# B&R Automation Studio project AriesV2 (part 3)

#### wbrPingSvc.c
```c
/********************************************************************
 * \copyright -- Piedmont Automation
 ********************************************************************
 * Program : wbrPingSvc
 * \file :   wbrPingSvc.c
 * \author : Blanton Radford
 * \date Created: June 22, 2015
 *******************************************************************/

#include <string.h>
// #include <bur/plctypes.h>

// #include  "wbrsprintf.h"
#include  "wbrPingSvc.h"

DINT  wbrPingSvcInit(struct wbrPingService_typ* p)
{
  p->fb.enable=  1;
  // p->fb.pHost=   (UDINT)"192.168.44.220";
  p->fb.pHost=   (UDINT)p->destIPAddr;
  p->fb.timeout= p->timeout;                                                    // If ping not successful within (timeout x 10)ms, error occurs

  p->logbookID= arlogBASE_USER_LOG_IDENT;         /// \todo   change to user net log from wbrNetSvc

  return  0;
}

static  char* errorTextLookup(UINT erNum, char* erText, UDINT erTextLen)
{
  // TODO: use table(s) in file(s) for holding error text instead of the code below

  switch(erNum)
  {
   case 32750:  wbrsnprintf(erText, erTextLen, "No response from station %%s within the specified time");
    break;
   case 32751:  wbrsnprintf(erText, erTextLen, "IP address %%s not resolvable");
    break;
   case 32752:  wbrsnprintf(erText, erTextLen, "Resource problem in system.  Could not create socket for pinging %%s");
    break;
   case 32799:  wbrsnprintf(erText, erTextLen, "System level error when pinging %%s");
    break;
   case 0xFFFE: wbrsnprintf(erText, erTextLen, "System ping function not enabled when pinging %%s");
    break;

   default:     wbrsnprintf(erText, erTextLen, "Something went wrong with error text lookup - erNum in table?");
    break;
  }

  return erText;
}

// void printErrorText(UINT erNum, char* errorText, args)  //  TODO: with variable args
// {
// }

static  void printErrorText(BOOL prependErNum, UINT erNum, char* message, UDINT msgLen, char* ipAddr)
{
  // char  erText[100]= "",      // Will contain error text with inserted format specifiers for custom arguments
        // erFmtd[100]= "";      // Will contain above text with error number prepended
  char  erText[msgLen],      // Will contain error text with inserted format specifiers for custom arguments - v0.11.0
        erFmtd[msgLen];      // Will contain above text with error number prepended

  if(prependErNum)
  {
    wbrsnprintf(erFmtd,                                                           // Used in next wbrsnprintf
              sizeof(erFmtd),
              "%d: %s",
              erNum,
              errorTextLookup(erNum, erText, sizeof(erText)));                  // Finds custom error text for error erNum

    wbrsnprintf(message,
              msgLen,
              erFmtd,                                                           // From wbrsnprintf above
              ipAddr);
    return;
  }

  // Else do not prepend error number
  wbrsnprintf(message,
            msgLen,
            errorTextLookup(erNum, erText, sizeof(erText)),                     // Finds custom error text for error erNum
            ipAddr);
  return;
}

/*! \brief Print the number of successes for debugging
    \pre   None
*/
static  char * printMsgSuccess(struct wbrPingService_typ* p)
{
  wbrsnprintf(  p->message                                                    // Print the number of successes for debugging
              , sizeof(p->message)
              , "Station %s pinged successfully %d times"
              , p->destIPPrev
              , p->count
              );
  return  p->message;
}

/*! \brief Print the number of failures for debugging
    \pre   None
*/
static  char * printMsgFailure(struct wbrPingService_typ* p)
{
  wbrsnprintf(  p->message1                                                    // Print the number of failures for debugging
              , sizeof(p->message1)
              , "Station %s ping failed %d times"
              , p->destIPPrev
              , p->count
              );
  return  p->message1;
}

DINT  wbrPingStation(struct wbrPingService_typ* p)
{
  if(!p->enable && !p->count)  return  0xFFFE;

  if(!p->enable){

    if(p->failed) requestMessageToLogDefault( (UDINT)printMsgFailure(p));
    else          requestMessageToLogDefault( (UDINT)printMsgSuccess(p));

    p->count=
        p->failed=
        p->errorStatus= 0;

    return  0xFFFE;
  }

  bgTimerCyclic(&p->retryTimer);

  if(!p->failed && p->retryTimer.IN && !p->retryTimer.Q)  return  0xFFFF;       // Return if success and the timer is running for the next attempt

  if(strcmp(p->destIPPrev, p->destIPAddr) )                                                               // new station
  {
    wbrsnprintf(p->message,                                                     // Print the number of failures for debugging
              sizeof(p->message),
              "Station %s is a new station",
              p->destIPAddr
              );
    requestMessageToLogDefault( (UDINT)p->message);

    if(p->failed) requestMessageToLogDefault( (UDINT)printMsgFailure(p));
    else          requestMessageToLogDefault( (UDINT)printMsgSuccess(p));

    p->count=
        p->failed=
        p->errorStatus= 0;
    wbrsnprintf(p->destIPPrev, sizeof(p->destIPPrev), p->destIPAddr);
  }

  p->fb.pHost=   (UDINT)p->destIPAddr;
  p->fb.timeout= p->timeout;

  IcmpPing(&p->fb);

  switch(p->fb.status)
  {
   case 0xFFFF:       //  busy
    // p->errorStatus= 0;
    return  0xFFFF;

   case 0:            //  success
    if(p->failed)                                                               // fail state changed from fail to success
    {
      requestMessageToLogDefault( (UDINT)printMsgFailure(p));
      p->count=
          p->failed=
          p->errorStatus= 0;
    }

    p->failed=  0;
    p->count++;
    bgTimerStart(&p->retryTimer, p->repeatTime);

    printMsgSuccess(p);

    if(!((p->count - 1) % p->successesToCount))
    {
      requestMessageToLogDefault( (UDINT)p->message);
    }
    return  0;

   case 32750:        // Defined error statuses
   case 32751:
   case 32752:
   case 32799:
   case 0xFFFE:
    printErrorText(1, p->fb.status, p->message, sizeof(p->message), p->destIPAddr);
    break;

   default:
    wbrsnprintf(p->message,
              sizeof(p->message),
              "%d: Should not get here when pinging IP address %s",
              p->fb.status,
              p->destIPAddr);
    break;
  }

  if(!p->failed || (p->fb.status != p->errorStatus)) //
  {
    p->errorStatus= p->fb.status;
    requestMessageToLog( (UDINT)p->message
                       , p->logbookID
                       , arlogLEVEL_INFO
                       , 55550
                       , (UDINT)&p->fb.status
                       , (UDINT)sizeof(p->fb.status)
                       );
    p->count= 0;
  }

  if(p->count == 1)
  {
    requestMessageToLog( (UDINT)"Current ping error is repeating"
                       , p->logbookID
                       , arlogLEVEL_INFO
                       , 55550
                       , (UDINT)&p->fb.status
                       , (UDINT)sizeof(p->fb.status)
                       );
  }

  p->failed=  1;
  p->count++;
  return  p->count;
}

// void  mbTCPdiag()
// {
  // slave.diag.ping.fb.pHost=   (UDINT)slave.diag.ping.destIPAddr;
  // if(slave.diag.ping.enable)   pingPeer(&slave.diag.ping, 512);
// }

DINT  wbrSQL_DT2_ISOFmtdStringFromDT(struct DTStructure * pDT, char * pDst, UDINT dstSize)
{
  return  wbrsnprintf(pDst, dstSize, "%04d-%02d-%02dT%02d:%02d:%02d",
                      pDT->year, pDT->month, pDT->day,
                      pDT->hour, pDT->minute, pDT->second);
}
```

### Library Logical/UserLibraries/wbrServices/wbrsprintf (ANSIC) - Writes user-formatted output to a string

#### wbrsprintf.h
```c
/*!
 ********************************************************************
### Library : wbrsprintf
 *  Package : WBRServices
 * \file :   wbrsprintf.h
 * \author : Blanton Radford
 * \date Created: May 3, 2016
 * \copyright -- Piedmont Automation
 *******************************************************************
 * \brief Header file for snprintf functions.
          Use of sprintf functions discouraged as snprintf is guaranteed to
          stop writing once buf_size is filled.
 ********************************************************************/

#include <stdarg.h>

/*! These are not included by default to strongly discourage the use of sprintf
    If they are uncommented, please uncomment the warning as well
*/
// #warning  "Consider using snprintf function for safety"
// int wbrvsprintf(char *s, const char *fmt, va_list ap);
// int  wbrsprintf(char *s, const char *fmt, ...);

int wbrvsnprintf(char *s, int buf_size, const char *fmt, va_list ap);
int  wbrsnprintf(char *s, int buf_size, const char *fmt, ...);
```

### Library Logical/UserLibraries/wbrServices/wbrSvcUtilities/wbrBytUtil (ANSIC)

#### wbrBytUtilities.c
```c
/*!
 ********************************************************************
### Library : wbrBytUtil
 * \file :   wbrBytUtilities.c
 * \author : Blanton Radford
 * \date Created: Friday, October 14, 2016
 * \copyright  Piedmont Automation
 ********************************************************************
 * \brief Utilities for extracting bytes from or packing bytes into words,
          ints, etc.
 ********************************************************************/

/*! \mainpage Example logbook manager to create, get info from, and write to user created logbooks using \e wbrLogSvc functions

#   A main heading

    Some text

##  A subheading

    More text

    A separator
    -----------

    Even more txt

##  See \e Files selection above for more info on the functions and how to
##  use them.
*/

#include "wbrBytUtil.h"

/*————————————————————————————————————————————————————————————————————————————*/
/*! \brief Get the high 16-bit word from a 32-bit double word
    \pre

rtyp  �(x)뿓뿓뿬  뿓뿓뿓뿓뿓뿓뾞rgument comments뿓뿓뿓뿓뿓뿓뿓뿓뿓뿓뿓뿓뿓뿓븬븰  */

UINT  getHiWord(

        UDINT dword                     //!< 32-bit unsigned int or word input
      )
{
 UINT hi=  (UINT)(dword >> 16);

  return  hi;
}
/*————————————————————————————————————————————————————————————————————————————*/

/*————————————————————————————————————————————————————————————————————————————*/
/*! \brief Split 32-bit Dword or integer into two 16-bit words
    \pre

rtyp              �(x)뿓뿓뿓뿓�  뾞rgument comments뿓뿓뿓뿓뿓뿓뿓뿓뿓뿓뿓뿓뿑븬�  */

dwordToWords_typ  dwordToWords(

        UDINT dword                     //!< 32-bit unsigned int or word input
      )
{
 dwordToWords_typ word;

  word.lo=  (UINT)dword;
  word.hi=  (UINT)(dword >> 16);

  return  word;
}
/*————————————————————————————————————————————————————————————————————————————*/

/*————————————————————————————————————————————————————————————————————————————*/
/*! \brief Split 16-bit Dword or integer into two 8-bit bytes
    \pre

rtyp              �(x)뿓뿓뿓뿬  뿓뿓뿓뿓뿓뿓뿓뿓뿓argument comments뿓뿓뿓뿓뿓뿓뿓뿑븬�  */

wordToBytes_typ   wordToBytes(

        UDINT word                     //!< 32-bit unsigned int or word input
      )
{
 wordToBytes_typ byte;

  byte.lo=  (UINT)word;
  byte.hi=  (UINT)(word >> 8);

  return  byte;
}
/*————————————————————————————————————————————————————————————————————————————*/
```

- Library Logical/UserLibraries/wbrServices/wbrSvcUtilities/wbrFltUtil (ANSIC) (no source held here)

### Library Logical/UserLibraries/jgLibs/jgLibC (ANSIC)
Depends on: standard, sys_lib, wbrLogSvc, MpAxis, Acp10par

#### VirtualDebounce.typ - Exported data types
```iecst
TYPE
	Debounce_Config_Struct : 	STRUCT
		Timer_On : REAL;
		Timer_Off : REAL;
	END_STRUCT;
END_TYPE
```

#### jgLibC.fun - Exported functions and function blocks
```iecst
FUNCTION Tms : UDINT
	VAR_INPUT
		in : REAL;
	END_VAR
END_FUNCTION

FUNCTION_BLOCK Debounce_Signal (*TODO: Add your comment here*) (*$GROUP=User,$CAT=User,$GROUPICON=User.png,$CATICON=User.png*)
	VAR_INPUT
		input : {REDUND_UNREPLICABLE} USINT;
		pConfigVals : REFERENCE TO Debounce_Config_Struct;
	END_VAR
	VAR_OUTPUT
		Signal_Debounced : USINT;
	END_VAR
	VAR
		Ton : TON;
		Tof : TOF;
	END_VAR
END_FUNCTION_BLOCK

FUNCTION_BLOCK FBK_Init_Logbook (*TODO: Add your comment here*) (*$GROUP=User,$CAT=User,$GROUPICON=User.png,$CATICON=User.png*)
	VAR_INPUT
		Enable : BOOL;
		Name : STRING[80];
	END_VAR
	VAR_OUTPUT
		pLog : UDINT;
	END_VAR
	VAR
		Logbook : wbrLogServiceLogbookInfo_typ;
		ii_init_calls : UDINT;
	END_VAR
END_FUNCTION_BLOCK
```

#### Debounce_Signal.c
```c
#include <bur/plctypes.h>

#include <jgLibC.h>

/* TODO: Add your comment here */
void Debounce_Signal(struct Debounce_Signal* p)
{

	if(p && p->pConfigVals){

		p->Ton.PT = Tms(p->pConfigVals->Timer_On);
		p->Tof.PT = Tms(p->pConfigVals->Timer_Off);

		p->Ton.IN = p->input;
		bgTimerCyclic(&p->Ton);
		p->Tof.IN = p->Ton.Q;
		bgTimerOffCyclic(&p->Tof);
		p->Signal_Debounced = p->Tof.Q;
	}
}
```

#### Tms.c
```c
/********************************************************************
 * COPYRIGHT -- Microsoft
 ********************************************************************
 * Library: jgLibC
 * File: Indexer_Helper_functions.c
 * Author: Admin
 * Created: May 11, 2015
 *******************************************************************/

#include <bur/plctypes.h>
#include <jgLibC.h>
UDINT Tms(REAL in){
	UDINT var_return = 0;

	var_return = (UDINT) (1000 * in);

	return var_return;
}
```

#### FBK_Init_Logbook.c
```c
#include <bur/plctypes.h>

#ifdef _DEFAULT_INCLUDES
#include <AsDefault.h>
#endif

#include <jgLibC.h>
#include <wbrsprintf.h>
/* TODO: Add your comment here */
void FBK_Init_Logbook(struct FBK_Init_Logbook* p)
{
//	return;

	if(!p->Enable) return;

	p->ii_init_calls = 0;

	wbrsnprintf(p->Logbook.name, sizeof(p->Logbook.name), p->Name);

	do {
		getLogbookInfo(&p->Logbook);
		p->ii_init_calls++;
	} while(p->Logbook.status == 0xFFFF && p->ii_init_calls <= MAX_CALLS_INIT_LOGBOOK);

	if(p->Logbook.status == arlogERR_NOTEXISTING){
		p->ii_init_calls = 0;
		do {
			createNewLogbook(&p->Logbook);
			p->ii_init_calls++;
		} while(p->Logbook.status == 0xFFFF && p->ii_init_calls <= MAX_CALLS_INIT_LOGBOOK);

		if(!p->Logbook.status){
			requestMessageToLog((UDINT) "Logbook Created", p->Logbook.ident, arlogLEVEL_INFO, 0, 0, 0);
		}
		else{
			requestMessageToLog((UDINT) "Logbook Creation Failed", arlogBASE_USER_LOG_IDENT, arlogLEVEL_INFO, (UDINT) p->Logbook.status, 0, 0);
		}

	}

	p->pLog = p->Logbook.ident;

	return;

}
```

### HW_modules.typ
```iecst
(********************************************************************
 * COPYRIGHT --
 ********************************************************************
 * File: Global.typ
 * Author: John
 * Created: January 18, 2015
 ********************************************************************
 * Global data types of project CNC_Lite
 ********************************************************************)

TYPE
	GenericKinetics_typ : 	STRUCT
		Distance : REAL;
		Position : REAL;
		Velocity : REAL;
		Acceleration : REAL;
		Deceleration : REAL;
		Direction : USINT;
		JogVelocity : REAL;
	END_STRUCT;
	DSP_Error_typ : 	STRUCT
		FifoEmpty : BOOL;
		FifoFull : BOOL;
		TargetTimeViolation : BOOL;
		FrequencyViolation : BOOL;
	END_STRUCT;
	X20DS1119_PosCtrl_typ : 	STRUCT
		iModuleOK : BOOL;
		iSDCLifeCount : SINT;
		oMoveEnable : BOOL;
		oMoveTargetPos : DINT;
		iMovePos : DINT;
		iCounterPosition : DINT;
		iR : BOOL;
	END_STRUCT;
	PAIDemoKitIO_typ : 	STRUCT
		DM1321 : X67DM1321_L12_1_typ;
		BT9400 : X20BT9400_typ;
		PLK_IF : Plk_IF_typ;
		DS1119 : X20DS1119_PosCtrl_typ;
	END_STRUCT;
	Plk_IF_typ : 	STRUCT
		iCycleCongestionCount : UDINT;
		iCycleIdleTime : UDINT;
		iCycleTimeViolationCount : UDINT;
		iFailedCycleCount : UDINT;
		iCycleCount : UDINT;
		iNettimeOffset : DINT;
		iNettimeSoC : DINT;
		iTimeNanoSeconds : UDINT;
		iTimeSeconds : UDINT;
		iSyncOK : BOOL;
		iCycleOK : BOOL;
		iNodeNumber : USINT;
		iOutputDMAMargin : DINT;
		iLinkOK : BOOL;
	END_STRUCT;
	X20AI1744_typ : 	STRUCT
		iModuleOk : BOOL;
		oOutputConfig : USINT;
		iStatusAI : USINT;
		iAI : DINT;
	END_STRUCT;
	X20BR9300_typ : 	STRUCT
		iModuleOk : BOOL;
		iStatusInput : ARRAY[0..1]OF BOOL;
	END_STRUCT;
	X20BT9100_typ : 	STRUCT
		iModuleOk : BOOL;
		iStatusInput : ARRAY[0..1]OF BOOL;
		iSupplyCurrent : USINT;
		iSupplyVoltage : USINT;
	END_STRUCT;
	X20BT9400_typ : 	STRUCT
		iModuleOk : BOOL;
		iStatusInput : ARRAY[0..1]OF BOOL;
		iSupplyCurrent : USINT;
		iSupplyVoltage : USINT;
	END_STRUCT;
	X20DC4395_typ : 	STRUCT
		iModuleOK : BOOL;
		iStaleData : BOOL;
		iAB_Enc_Val : ARRAY[0..3]OF DINT;
		iPowerSupply : BOOL;
		oRefMode : USINT;
		iStatusABR : USINT;
	END_STRUCT;
	X20DI9372_typ : 	STRUCT
		iDI : ARRAY[0..11]OF BOOL;
		iModuleOk : BOOL;
	END_STRUCT;
	X20DO9322_typ : 	STRUCT
		iModuleOk : BOOL;
		iStatusDO : ARRAY[0..11]OF BOOL;
		oDO : ARRAY[0..11]OF BOOL;
	END_STRUCT;
	X20DS1119_typ : 	STRUCT
		iModuleOK : BOOL;
		iStaleData : BOOL;
		iSDCLifeCnt : SINT;
		iProtocolError : UINT;
		iProtocolSequenceViolation : UINT;
		iPowerSupply : ARRAY[0..1]OF BOOL;
		oMoveEnable : BOOL;
		oMoveTargetTime : INT;
		oMoveTargetPosition : DINT;
		iMovePosition : DINT;
		iMoveTimeValid : INT;
		oError : DSP_Error_typ;
		iError : DSP_Error_typ;
	END_STRUCT;
END_TYPE

(*Insert your comment here.*)

TYPE
	X67DM1321_L12_1_typ : 	STRUCT
		iModuleOK : BOOL;
		oDigitalOutput : ARRAY[0..15]OF BOOL;
		iStatusDigitalOutput : ARRAY[0..15]OF BOOL;
	END_STRUCT;
	X20SLX910_typ : 	STRUCT
		iModuleOK : BOOL;
	END_STRUCT;
	X20DM9324_typ : 	STRUCT
		iModuleOK : BOOL;
	END_STRUCT;
	X20CM8281_typ : 	STRUCT
		iModuleOK : BOOL;
	END_STRUCT;
	X20DOF322_typ : 	STRUCT
		iModuleOK : BOOL;
	END_STRUCT;
	X20DIF371_typ : 	STRUCT
		iModuleOK : BOOL;
	END_STRUCT;
	X20BC0083_typ : 	STRUCT
		iModuleOK : BOOL;
		iSerialNumber : UDINT;
		iModuleID : UINT;
		iHWVariant : UINT;
		iFirmwareVersion : UINT;
		iEthRxLost : DINT;
		iEthRxOverSize : DINT;
		iEthRxCRCErr : DINT;
		iEthRxOverflow : DINT;
		iEthTxCollision : DINT;
		iEthPhy1LinkOK : BOOL;
		iEthPhy1LinkLoss : DINT;
		iEthPhy2LinkOK : BOOL;
		iEthPhy2LinkLoss : DINT;
		iNetTime : DINT;
	END_STRUCT;
	X20CS1030_typ : 	STRUCT
		iModuleOK : BOOL;
		iSerialNumber : UDINT;
		iModuleID : UINT;
		iHWVariant : UINT;
		iFirmwareVersion : UINT;
	END_STRUCT;
	X20PD2113_typ : 	STRUCT
		iModuleOK : BOOL;
		iSerialNumber : UDINT;
		iModuleID : UINT;
		iHWVariant : UINT;
		iFirmwareVersion : UINT;
		iStatusFuse : BOOL;
		iPowerSupply : BOOL;
	END_STRUCT;
	X20PS9400_typ : 	STRUCT
		iModuleOK : BOOL;
		iSerialNumber : UDINT;
		iModuleID : UINT;
		iHWVariant : UINT;
		iFirmwareVersion : UINT;
		iStatusInput1 : BOOL;
		iStatusInput2 : BOOL;
	END_STRUCT;
	X20SM1436_typ : 	STRUCT
		iModuleOK : BOOL;
		iStaleData : BOOL;
		iSerialNumber : UDINT;
		iModuleID : UINT;
		iHWVariant : UINT;
		iFirmwareVersion : UINT;
		iLifeCount : SINT;
		oSetTime : INT;
		oMotor1Step : INT;
		oDriveEnable : BOOL;
		oBoostCurrent : BOOL;
		oStandStillCurrent : BOOL;
		oClearError : BOOL;
		iDriveOK : BOOL;
		iStallError : BOOL;
		iTempError : BOOL;
		iCurrentError : BOOL;
		iOverCurrentError : BOOL;
		iActPos : INT;
		iRefPulsePos : INT;
		iRefPulsCount : SINT;
		iEncOK : BOOL;
		iActTime : INT;
		iTriggerTime : INT;
		iTriggerCount : SINT;
		iStatusInput : ARRAY[0..3]OF BOOL;
		iModPowerSupplyError : BOOL;
	END_STRUCT;
	X20SO4110_typ : 	STRUCT
		iModuleOK : BOOL;
		iSerialNumber : UDINT;
		iModuleID : UINT;
		iHWVariant : UINT;
		iFirmwareVersion : UINT;
	END_STRUCT;
END_TYPE
```

### Library Logical/UserLibraries/jgLibs/VA_Setup

#### VA_Setup.fun
```iecst
FUNCTION VA_SetupSt : UINT
VAR_INPUT
		enable	:BOOL;
		VcHandle	:REFERENCE TO UDINT;
		pProjectName	:STRING[9];
	END_VAR
END_FUNCTION
```

#### va_setup.c
```c
#include <bur/plc.h>
#include <bur/plctypes.h>
#include <visapi.h>

unsigned short VA_SetupSt(plcbit enable, unsigned long* VcHandle, plcstring* pProjectName)
{
    return VA_SetupX(enable,(UDINT)(VCHANDLE*)VcHandle,pProjectName);
}
```

### IO.typ - not listed in the package file held
```iecst
TYPE
	IO_Status_typ : 	STRUCT
		iEmergencyStopStatus_3SB1A_I00 : BOOL;
		iBatteryPresent_3BF7A_I06 : BOOL;
		oFolderInsertOKLight_6HL1E_U16 : USINT;
		oWarningLightAlarm_6HL2E_U17 : USINT;
		New_Member : USINT;
		New_Member5 : USINT;
		New_Member4 : USINT;
		New_Member3 : USINT;
		New_Member2 : USINT;
	END_STRUCT;
	IO_Buttons_typ : 	STRUCT
		iStart_3SB3A_I02 : USINT;
		iStop_3SB4A_I03 : USINT;
		iReset_3SB5A_I04 : USINT;
		New_Member1 : USINT;
		New_Member : USINT;
		New_Member5 : USINT;
		New_Member4 : USINT;
		New_Member3 : USINT;
		New_Member2 : USINT;
	END_STRUCT;
	IO_Motor_typ : 	STRUCT
		iMotorInhibitStatus_SM1_I05 : BOOL;
		iBladeEngineTravelStop_3SQ8A_I07 : BOOL;
		iDriveOK_4KA4B_I11 : USINT;
		iBladeStartSignal_4SB5A_I12 : USINT;
		iRollerStartSignal_4SB6A_I13 : USINT;
		oCreasingEngineContactor_SM1_U23 : USINT;
	END_STRUCT;
	IO_Control_typ : 	STRUCT
		iCreaseSelector_3SA2A_I01 : USINT;
		iAutoModeSelector_4SA2A_I09 : USINT;
		iManualModeSelector_4SA2AI10 : USINT;
		oDriveEnable_3SB1A_U20 : USINT;
		New_Member1 : USINT;
	END_STRUCT;
	CMA_Arimat_IO_typ : 	STRUCT
		Button : IO_Buttons_typ;
		Status : IO_Status_typ;
		Motor : IO_Motor_typ;
		Control : IO_Control_typ;
		New_Member3 : USINT;
		New_Member2 : USINT;
		New_Member1 : USINT;
		New_Member : USINT;
	END_STRUCT;
END_TYPE
```

### varPkg.var - not listed in the package file held
```iecst
(*<--------------------------------------------->*)
(*Pre-compile Constants*)
VAR CONSTANT
	MAX_IDX_CREASES : UDINT := 19;
END_VAR
(*<--------------------------------------------->*)
(*IO Values*)
VAR
	IO : CMA_Arimat_IO_typ;
END_VAR
(*<--------------------------------------------->*)
(*Control State Machine States*)
VAR
	MachineState : CMA_Arimat_MachineState_Enum;
	ProcessState : CMA_Arimat_PrcsState_Enum;
END_VAR
(*<--------------------------------------------->*)
(*<--------------------------------------------->*)
(**)
(*<--------------------------------------------->*)
(*<--------------------------------------------->*)
(**)
(*<--------------------------------------------->*)
(*Insert your comment here.*)
(*Insert your comment here.*)
(*Insert your comment here.*)
(*Insert your comment here.*)
```

### Library Logical/Application_Logic/lib5200 (IEC)
Depends on: libDisp, libInsp

#### RecCfg.typ
```iecst
TYPE
	Generic_Cfg_HMI_typ : 	STRUCT
		passwordSetup : STRING[15];
		passwordEngineer : STRING[15];
		passwordFactory : STRING[15];
		Disp_Trend_SampleCount : UDINT;
		MuteSwitchBypassTO : REAL;
		Access_Level_Cfg : UDINT;
		Access_Level_Recipe : UDINT;
		Access_Level_ForceIO : UDINT;
		Access_Level_HomeForce : UDINT;
		Access_Level_FileIO : UDINT;
		Admin_Limit_Run_Velocity : REAL;
		LoginTO_S : REAL;
		MachineLang : UDINT;
	END_STRUCT;
	HERNON_Cfg_Mechanics_typ : 	STRUCT
		I_Motor_Sprocket_Gear_Ratio : UDINT;
		N_Sprocket_Teeth : UDINT;
		N_VBlocks_Belt_Total : UDINT;
	END_STRUCT;
	Global_Rec_typ : 	STRUCT
		MagicPrefix : UDINT;
		Dispense : ARRAY[0..MAX_IDX_DISPENSE_UNITS]OF HERNON_Rec_Dispense_typ;
		Inspect : ARRAY[0..MAX_IDX_INSPECT_UNITS]OF HERNON_Rec_Inspect_typ;
		MagicSuffix : UDINT;
	END_STRUCT;
	Global_Cfg_typ : 	STRUCT
		MagicPrefix : UDINT;
		Dispense : ARRAY[0..MAX_IDX_DISPENSE_UNITS]OF HERNON_Cfg_Dispense_typ;
		Inspect : ARRAY[0..MAX_IDX_INSPECT_UNITS]OF HERNON_Cfg_Inspect_typ;
		Mechanics : HERNON_Cfg_Mechanics_typ;
		HMI : {REDUND_UNREPLICABLE} Generic_Cfg_HMI_typ;
		MagicSuffix : UDINT;
	END_STRUCT;
END_TYPE
```

### Library Logical/Application_Logic/pkgDispense/Dispense

#### Types.typ
```iecst
TYPE
	HERNON_DISP_REASONS_ENUM :
		(
		DISPENSE_SINGLE_SHOT := 0,
		DISPENSE_PURGE := 1
		);
	HERNON_Dispense_Unit_ID_Enum :
		(
		DISPENSE_PRIMER := 0,
		DISPENSE_MOUTH := 1
		);
	HERNON_Disp_AppTimers_typ : 	STRUCT
		Max_Valve_NotRdy_NegEdge : TON;
		Max_Time_Disp_Output_NegEdge : TON;
		Max_Valve_Rdy_Reset : TON;
		Max_Dispense_Output_High : TON;
	END_STRUCT;
	HERNON_Dispense_App_typ : 	STRUCT
		VBlock_At_Dispense_Unit : UDINT;
		VBlock_Fract_Pos : REAL;
		Flag_Dispense_Purge_Now : BOOL;
		Flag_Dispense_Trigger_Now : BOOL;
		DispState : HERNON_Dispense_Enum;
		ii_Trend_Idx_DP : UDINT;
		Disp_Single_Shot_Or_Purge : HERNON_DISP_REASONS_ENUM;
		Edge_Reading_At_Disp_Trigger : DINT;
		Timer : HERNON_Disp_AppTimers_typ;
		ii_shot_counter : UDINT;
	END_STRUCT;
END_TYPE
```

#### Variables.var
```iecst
VAR
	ii_dispense_units : UDINT;
END_VAR
(*Insert your comment here.*)
VAR
	FBK_Disp_Valve : ARRAY[0..MAX_IDX_DISPENSE_UNITS] OF HernonDispValve;
	Init_Logbook : FBK_Init_Logbook;
END_VAR
```

#### libDisp.fun
```iecst
FUNCTION_BLOCK HernonDispValve (*TODO: Add your comment here*) (*$GROUP=User,$CAT=User,$GROUPICON=User.png,$CATICON=User.png*)
	VAR_INPUT
		pDispVBlock : REFERENCE TO VBlock_Object_typ;
		pDispRec : REFERENCE TO HERNON_Rec_Dispense_typ;
		pDispCfg : REFERENCE TO HERNON_Cfg_Dispense_typ;
		pDispenseIO : REFERENCE TO HERNON_Inline_Dispense_Item_typ;
		pMechanics : REFERENCE TO HERNON_Cfg_Mechanics_typ;
		iNettime : DINT;
		MachineState : Global_State_Enum;
		VBlock_Fractional_Position : REAL;
		Current_VBlock_At_PiP_Sensor : UDINT;
		idx_disp_unit : USINT;
	END_VAR
	VAR
		DispVar : HERNON_Dispense_App_typ;
		DispVar_LastCycle : HERNON_Dispense_App_typ;
		Alarms : HERNON_Alarm_Dispense_typ;
	END_VAR
END_FUNCTION_BLOCK
```

#### HernonDispValve.st
```iecst
(* TODO: Add your comment here *)
FUNCTION_BLOCK HernonDispValve

	DispVar.VBlock_At_Dispense_Unit := (Current_VBlock_At_PiP_Sensor + (pMechanics.N_VBlocks_Belt_Total - pDispCfg.VBlock_Offset_From_PiP_Sensor)) MOD (pMechanics.N_VBlocks_Belt_Total);
	DispVar.VBlock_Fract_Pos := VBlock_Fractional_Position;

	IF pDispRec.Enable = 1 AND DispVar.VBlock_At_Dispense_Unit <> DispVar_LastCycle.VBlock_At_Dispense_Unit AND pDispVBlock.VBlock_Is_Occupied THEN
		DispVar.Flag_Dispense_Trigger_Now := TRUE;
		pDispVBlock.Dispense[idx_disp_unit].Dispense_Has_Been_Triggered[DispVar.ii_shot_counter] := TRUE;
	END_IF;

	//TODO: Return SM to INIT here on Stop/Reset Requested?

	IF NOT pDispenseIO.EdgeGen.iEdgeGenWarning THEN
		pDispenseIO.EdgeGen.oQuitEdgeGenWarning := FALSE;
	END_IF;

	IF NOT pDispenseIO.EdgeGen.iEdgeGenError THEN
		pDispenseIO.EdgeGen.oQuitEdgeGenError := FALSE;
	END_IF;

	CASE DispVar.DispState OF
		DISPENSE_STATE_INIT:
			pDispenseIO.oDispTrigger := FALSE;
			DispVar.Flag_Dispense_Trigger_Now := FALSE;
			DispVar.ii_shot_counter := 0;
			pDispenseIO.EdgeGen.oEnableEdgeGen := TRUE;

			IF pDispenseIO.EdgeGen.iEdgeGenError AND pDispenseIO.EdgeGen.oQuitEdgeGenError THEN
				pDispenseIO.EdgeGen.oQuitEdgeGenError := TRUE;
			ELSE
				pDispenseIO.EdgeGen.oQuitEdgeGenError := FALSE;
			END_IF;

			IF pDispenseIO.EdgeGen.iEdgeGenWarning AND pDispenseIO.EdgeGen.oQuitEdgeGenWarning THEN
				pDispenseIO.EdgeGen.oQuitEdgeGenWarning := TRUE;
			ELSE
				pDispenseIO.EdgeGen.oQuitEdgeGenWarning := FALSE;
			END_IF;

			IF pDispRec.Enable = 0 THEN
				DispVar.DispState := DISPENSE_STATE_DISABLED;
			ELSIF (pDispenseIO.iValveReady AND NOT pDispenseIO.EdgeGen.iEdgeGenError) THEN
				DispVar.DispState := DISPENSE_STATE_READY;
			END_IF;

		DISPENSE_STATE_READY:
			IF (NOT pDispenseIO.iValveReady OR pDispenseIO.EdgeGen.iEdgeGenError) AND (MachineState = gSTATE_START_REQUESTED OR MachineState = gSTATE_RUNNING) THEN
//				pDispVBlock.Error.DispenseValveError := TRUE;
				Alarms.Valve_Error_1 := TRUE;

				DispVar.DispState := DISPENSE_STATE_ERROR;
			ELSIF DispVar.Flag_Dispense_Trigger_Now THEN
				//Reset HMI trend datapoints
//				brsmemset(ADR(pDispVCTrend.iValveReady[0]), 0, MAX_IDX_DISPENSE_VC_ARRAY + 1);
//				brsmemset(ADR(pDispVCTrend.oDispTrigger[0]), 0, MAX_IDX_DISPENSE_VC_ARRAY + 1);
//				brsmemset(ADR(pDispVCTrend.iReadOutputStatus[0]), 0, MAX_IDX_DISPENSE_VC_ARRAY + 1);
				DispVar.ii_Trend_Idx_DP := 0;
				//
				DispVar.ii_shot_counter := 0;
				pDispenseIO.oDispTrigger := TRUE;
				bgTimerStart(DispVar.Timer.Max_Valve_NotRdy_NegEdge, Tms(pDispCfg.Disp_Valve_Max_RDY_NegEdge_S));

				DispVar.Edge_Reading_At_Disp_Trigger := pDispenseIO.EdgeGen.iEdgeMasterTime;//Nearly lost my mind to this one, need to document edge reading immediately before triggering output, as the high-speed edge detector has no debounce and it can possibly be a "dirty switch"
				DispVar.Flag_Dispense_Trigger_Now := FALSE;
				DispVar.Disp_Single_Shot_Or_Purge := DISPENSE_SINGLE_SHOT;
				DispVar.DispState := DISPENSE_STATE_WAIT_VALVE;
			ELSIF DispVar.Flag_Dispense_Purge_Now THEN
				pDispenseIO.oDispTrigger := TRUE;

				bgTimerStart(DispVar.Timer.Max_Dispense_Output_High, Tms(pDispCfg.Disp_Valve_Max_Output_High_TO_S));
				DispVar.Edge_Reading_At_Disp_Trigger := pDispenseIO.EdgeGen.iEdgeMasterTime;

				DispVar.Disp_Single_Shot_Or_Purge := DISPENSE_PURGE;
				DispVar.DispState := DISPENSE_STATE_DISPENSING;
			END_IF;

		DISPENSE_STATE_WAIT_VALVE:
			IF pDispenseIO.EdgeGen.iEdgeMasterTime <> DispVar.Edge_Reading_At_Disp_Trigger THEN
				pDispenseIO.oDispTrigger := FALSE;
				//Incrementing the edge gen sequence number is what causes the new timestamp to take hold (otherwise, it would trigger every time the clock rolls over)
				pDispenseIO.EdgeGen.oEdgeGenTimestamp := pDispenseIO.EdgeGen.iEdgeMasterTime + Tms(pDispRec.Disp_Valve_Edgemode_Pulse_TO_ms);//Yeah, this looks wrong, but it's probably right.
				pDispenseIO.EdgeGen.oEdgeGenSequence := pDispenseIO.EdgeGen.oEdgeGenSequence + 1;
				//Timer for maximum amount of time to wait before throwing an error, since the DO is reset via the edge generator and not the IO BOOL datapoint itself
				bgTimerStart(DispVar.Timer.Max_Time_Disp_Output_NegEdge, REAL_TO_UDINT(pDispRec.Disp_Valve_Edgemode_Pulse_TO_ms) + Tms(pDispCfg.Disp_Output_NegEdge_Margin_S));
				//
				DispVar.DispState := DISPENSE_STATE_DISPENSING;
			ELSIF (bgTimerIsTimeOut(DispVar.Timer.Max_Valve_NotRdy_NegEdge)) AND pDispenseIO.iValveReady THEN
				pDispenseIO.oDispTrigger := FALSE;

				pDispenseIO.EdgeGen.oEdgeGenTimestamp := iNettime + 10000;//Yeah, this looks wrong, but it's probably right.
				pDispenseIO.EdgeGen.oEdgeGenSequence := pDispenseIO.EdgeGen.oEdgeGenSequence + 1;//Incrementing the edge gen sequence number is what causes the new timestamp to take hold (otherwise, it would trigger every time the clock rolls over)

				Alarms.Dispense_ValveRdy_NegEdge_Err := TRUE;
				DispVar.DispState := DISPENSE_STATE_ERROR;
			END_IF;

		DISPENSE_STATE_DISPENSING:
			CASE DispVar.Disp_Single_Shot_Or_Purge OF
				DISPENSE_SINGLE_SHOT:
					IF NOT pDispenseIO.EdgeGen.iReadOutputStatus THEN
						bgTimerStart(DispVar.Timer.Max_Valve_Rdy_Reset, Tms(pDispCfg.Disp_Signal_Reset_MaxTO_S));
						DispVar.DispState := DISPENSE_STATE_WAIT_RESET;
					ELSIF bgTimerIsTimeOut(DispVar.Timer.Max_Time_Disp_Output_NegEdge) THEN
						Alarms.Disp_Output_Not_Reset := TRUE;
						DispVar.DispState := DISPENSE_STATE_ERROR;
					END_IF;
				DISPENSE_PURGE:
					pDispenseIO.oDispTrigger := FALSE;
					IF NOT DispVar.Flag_Dispense_Purge_Now THEN
						pDispenseIO.EdgeGen.oEdgeGenTimestamp := iNettime + 10000;//Yeah, this looks wrong, but it's probably right.
						pDispenseIO.EdgeGen.oEdgeGenSequence := pDispenseIO.EdgeGen.oEdgeGenSequence + 1;

						bgTimerStart(DispVar.Timer.Max_Valve_Rdy_Reset, Tms(pDispCfg.Disp_Signal_Reset_MaxTO_S));
						DispVar.DispState := DISPENSE_STATE_WAIT_RESET;
					ELSIF bgTimerIsTimeOut(DispVar.Timer.Max_Dispense_Output_High) THEN
						pDispenseIO.EdgeGen.oEdgeGenTimestamp := iNettime + 10000;//Yeah, this looks wrong, but it's probably right.
						pDispenseIO.EdgeGen.oEdgeGenSequence := pDispenseIO.EdgeGen.oEdgeGenSequence + 1;

						bgTimerStart(DispVar.Timer.Max_Valve_Rdy_Reset, Tms(pDispCfg.Disp_Signal_Reset_MaxTO_S));
						DispVar.DispState := DISPENSE_STATE_WAIT_RESET;
					END_IF;
			END_CASE;

		DISPENSE_STATE_WAIT_RESET://Wait for dispense valve ready to read back TRUE before the SM can go back into ready state, otherwise the rest of the code could trigger it too soon.
			IF pDispenseIO.iValveReady AND NOT DispVar.Flag_Dispense_Purge_Now THEN
				DispVar.ii_shot_counter := DispVar.ii_shot_counter + 1;

				IF DispVar.ii_shot_counter > pDispRec.Extra_Shots_Per_VBlock (*pDispCfg.Extra_Shots_Per_VBlock*) THEN
					DispVar.DispState := DISPENSE_STATE_READY;
				ELSE
					IF DispVar.VBlock_Fract_Pos < pDispRec.Vblock_Offset_Additional_Shots[DispVar.ii_shot_counter - 1] THEN
						DispVar.DispState := DISPENSE_STATE_WAIT_ADDITIONAL;
					ELSE
						Alarms.VBlock_Offset_Invalid := TRUE;
						DispVar.DispState := DISPENSE_STATE_ERROR;
					END_IF;
				END_IF;
			ELSIF bgTimerIsTimeOut(DispVar.Timer.Max_Valve_Rdy_Reset) AND (MachineState = gSTATE_START_REQUESTED OR MachineState = gSTATE_RUNNING) THEN
				Alarms.ValveRdy_Not_Reset := TRUE;
				DispVar.DispState := DISPENSE_STATE_ERROR;
			END_IF;

		DISPENSE_STATE_WAIT_ADDITIONAL:
			IF DispVar.VBlock_Fract_Pos > pDispRec.Vblock_Offset_Additional_Shots[DispVar.ii_shot_counter - 1] THEN
				pDispenseIO.oDispTrigger := TRUE;
				bgTimerStart(DispVar.Timer.Max_Valve_NotRdy_NegEdge, Tms(pDispCfg.Disp_Valve_Max_RDY_NegEdge_S));
				DispVar.Edge_Reading_At_Disp_Trigger := pDispenseIO.EdgeGen.iEdgeMasterTime;
				DispVar.Flag_Dispense_Trigger_Now := FALSE;
				DispVar.Disp_Single_Shot_Or_Purge := DISPENSE_SINGLE_SHOT;
				DispVar.DispState := DISPENSE_STATE_WAIT_VALVE;
			ELSIF DispVar.VBlock_At_Dispense_Unit <> DispVar_LastCycle.VBlock_At_Dispense_Unit THEN
				Alarms.VBlock_idx_during_shot_wait := TRUE;
				DispVar.DispState := DISPENSE_STATE_ERROR;
			END_IF;

		DISPENSE_STATE_DISABLED:
			IF pDispRec.Enable = 1 THEN
				DispVar.DispState := DISPENSE_STATE_INIT;
			END_IF;

		DISPENSE_STATE_ERROR:
		//State is exited via the event handler directly above state machine!
	END_CASE;

	bgTimerCyclic(DispVar.Timer.Max_Valve_NotRdy_NegEdge);
	bgTimerCyclic(DispVar.Timer.Max_Time_Disp_Output_NegEdge);
	bgTimerCyclic(DispVar.Timer.Max_Valve_Rdy_Reset);
	bgTimerCyclic(DispVar.Timer.Max_Dispense_Output_High);

	DispVar_LastCycle := DispVar;

END_FUNCTION_BLOCK
```

#### Main.st
```iecst
//     __ __                         __  ___               ___         __           _             ____
//    / // /__ _______  ___  ___    /  |/  /__ ____  __ __/ _/__ _____/ /___ ______(_)__  ___ _  /  _/__  ____
//   / _  / -_) __/ _ \/ _ \/ _ \  / /|_/ / _ `/ _ \/ // / _/ _ `/ __/ __/ // / __/ / _ \/ _ `/ _/ // _ \/ __/
//  /_//_/\__/_/ /_//_/\___/_//_/ /_/  /_/\_,_/_//_/\_,_/_/ \_,_/\__/\__/\_,_/_/ /_/_//_/\_, / /___/_//_/\__(_)
//                                                                                      /___/
//  Copyright

PROGRAM _INIT
	Init_Logbook.Enable := TRUE;
	Init_Logbook.Name := 'usr_disp';
	Init_Logbook();

	gHMITable_Rec_Dispense	(tableName := 'REC_DISPENSE',		nameSpace := 'hmiTable/Rec/Dispense',	Logbook := Init_Logbook.pLog, 		pOverallStats := ADR(gTableStats.Overall));
	gHMITable_Cfg_Dispense	(tableName := 'CFG_DISPENSE',		nameSpace := 'hmiTable/Cfg/Dispense',	Logbook := Init_Logbook.pLog, 		pOverallStats := ADR(gTableStats.Overall));

	FBK_Disp_Valve[0].pDispVBlock := ADR(gMachine.Belt.Mailbox[gMachine.Belt.Dispense[0].Current_VBlock_At_Dispense]);
	FBK_Disp_Valve[0].pDispRec := ADR(gRecCfg.active.Rec.Dispense[0]);
	FBK_Disp_Valve[0].pDispCfg := ADR(gRecCfg.active.Cfg.Dispense[0]);
	FBK_Disp_Valve[0].pDispenseIO := ADR(gMachine.IO.Dispense.Projectile);
	FBK_Disp_Valve[0].pMechanics  := ADR(gRecCfg.active.Cfg.Mechanics);
	FBK_Disp_Valve[0].idx_disp_unit := 0;
END_PROGRAM

PROGRAM _CYCLIC

//	FBK_Disp_Valve[0].iNettime
//	FBK_Disp_Valve[0].MachineState
//	FBK_Disp_Valve[0].VBlock_Fractional_Position
//	FBK_Disp_Valve[0].Current_VBlock_At_PiP_Sensor
	FBK_Disp_Valve[0]();

END_PROGRAM

PROGRAM _EXIT
	(* Insert code here *)

END_PROGRAM
```

### Disp_Belt_Types.typ
```iecst
TYPE
	HERNON_Belt_Disp_typ : 	STRUCT
		Current_VBlock_At_Dispense : UDINT;
		DispState : HERNON_Dispense_Enum;
	END_STRUCT;
END_TYPE
```

### Disp_StateMachine_States.typ
```iecst
TYPE
	HERNON_Dispense_Enum :
		(
		DISPENSE_STATE_INIT := 0,
		DISPENSE_STATE_READY := 1,
		DISPENSE_STATE_DISPENSING := 2,
		DISPENSE_STATE_WAIT_RESET := 3,
		DISPENSE_STATE_DISABLED := 4,
		DISPENSE_STATE_ERROR := 5,
		DISPENSE_STATE_WAIT_VALVE := 6,
		DISPENSE_STATE_WAIT_ADDITIONAL := 7,
		DISPENSE_STATE_MANUAL := 8
		);
END_TYPE
```

### Constants.var
```iecst
VAR CONSTANT
	MAX_IDX_MULTIPLE_DISPENSE_SHOTS : UDINT := 3;
END_VAR
```

### Program Logical/Application_Logic/pkgInspect/Inspect (IEC) - Manage all inspection related functionality

#### Types.typ
```iecst
TYPE
	HERNON_Inspect_Timers_typ : 	STRUCT
		Timer_Inspection_Trigger_DO_High : TON;
		Timer_Inspection_Illum_DO_High : TON;
		Timer_Inspection_Results_Wait : TON;
		Timer_Inspection_Trigger_Wait : TON;
		Timer_Max_Insp_Busy_Signal : TON;
	END_STRUCT;
	HERNON_Inspect_App_typ : 	STRUCT
		VBlock_At_Inspect_Unit : UDINT;
		Flag_Inspect_Trigger_Now : BOOL;
		Status : HERNON_Inspect_Enum;
		ii_VC_Trend_idx : UDINT;
		Timer : HERNON_Inspect_Timers_typ;
		VBlock_Fract_Pos : REAL;
	END_STRUCT;
END_TYPE
```

### Package Logical/paiComponents - pai Components and Libraries


- Library Logical/paiComponents/Libraries/sprintf2 (ANSIC) - A sprintf function implemenation (no source held here)

### Package Logical/paiComponents/bglib - pai C utilities

### bgdebugV2.h
```c
#ifndef _BG_DEBUG_H
#define _BG_DEBUG_H

#include <bur/plctypes.h>
#ifdef _DEFAULT_INCLUDES
	#include <AsDefault.h>
#endif

#ifdef WIN32
#define DBG printf
#define DBGMSG printf

#define DBGCRT printf
#define DBGERR printf
#define DBGWAR printf
#define DBGINF printf
#define DBGDBG printf

#else

#include <bur/plc.h>
#include "bgringbuffer.h"

#define BG_DEBUG_LEVEL_CRITICAL		0
#define BG_DEBUG_LEVEL_ERROR		1
#define BG_DEBUG_LEVEL_WARNING		2
#define BG_DEBUG_LEVEL_INFO			3
#define BG_DEBUG_LEVEL_DEBUG		4

#define BG_DEBUG_UNUSED	0x0

/*
- To completly remove debug msgs from the source code use:
#define BG_DEBUG_ENABLE 0
*/
#define BG_DEBUG_ENABLE 1

#if BG_DEBUG_ENABLE == 1
/*BG_DEBUG_ENABLE == 1 => debug messages present in the source code*/
#define DBG(pRB, format, args...)	bgRingBuffPutDbgInfo(pRB, __FILE__, (char*)__FUNCTION__, BG_DEBUG_LEVEL_CRITICAL, BG_DEBUG_UNUSED, format, ## args);
#define DBGMSG(pRB, format, args...)  {char txt[512]; snprintf2(txt, 512, format, ## args);	brsstrcat((UDINT)txt, (UDINT)"\r"); bgRingBuffPutString(pRB, txt);}

#define DBGCRT(pRB, format, args...)	bgRingBuffPutDbgInfo(pRB, __FILE__, (char*)__FUNCTION__, BG_DEBUG_LEVEL_CRITICAL, BG_DEBUG_UNUSED, format, ## args);
#define DBGERR(pRB, format, args...)	bgRingBuffPutDbgInfo(pRB, __FILE__, (char*)__FUNCTION__, BG_DEBUG_LEVEL_ERROR, BG_DEBUG_UNUSED, format, ## args);
#define DBGWAR(pRB, format, args...)	bgRingBuffPutDbgInfo(pRB, __FILE__, (char*)__FUNCTION__, BG_DEBUG_LEVEL_WARNING, BG_DEBUG_UNUSED, format, ## args);
#define DBGINF(pRB, format, args...)	bgRingBuffPutDbgInfo(pRB, __FILE__, (char*)__FUNCTION__, BG_DEBUG_LEVEL_INFO, BG_DEBUG_UNUSED, format, ## args);
#define DBGDBG(pRB, format, args...)	bgRingBuffPutDbgInfo(pRB, __FILE__, (char*)__FUNCTION__, BG_DEBUG_LEVEL_DEBUG, BG_DEBUG_UNUSED, format, ## args);

#else
/*BG_DEBUG_ENABLE == 0 => all debug messages removed from the source code*/
#define DBG(pRB, format, args...)  ;
#define DBGMSG(pRB, format, args...)  ;

#define DBGCRT(pRB, format, args...)	;
#define DBGERR(pRB, format, args...)	;
#define DBGWAR(pRB, format, args...)	;
#define DBGINF(pRB, format, args...)	;
#define DBGDBG(pRB, format, args...)	;

#endif /*#if BG_DEBUG_ENABLE*/

#endif /*#ifdef WIN32*/

#endif /*#ifndef _BG_DEBUG_H*/
```

### bgPVSerializeJSON.h
```c
/**\file: bgPVSerialize.h
*Serialize/deserialize a PV to/from text stream.
*/
#ifndef _BG_PVSERIALIZEJSON_H
#define _BG_PVSERIALIZEJSON_H

/**
Serialize a PV (*pvNameRoot) to an output stream (* toOutStream) with a max length of (lengthOutStream).
\param pvNameRoot ptr to a PV name
\param toOutStream ptr to an output stream (i.e. char buffer)
\param lengthOutStream max length of the output stream in bytes
\return -1 error
\return >=0 number of bytes written to the output stream
*/
DINT bgPVStructSerializeJSON(char* pvNameRoot, char* toOutStream, UDINT lengthOutStream);

/**
Deserialize a PV (*pvNameRoot) from an input stream (* fromStream) that contains (lengthStream) of valid text data.
\param pvNameRoot ptr to a PV name
\param fromStream ptr to an input stream (i.e. char buffer)
\param lengthStream length of the content in the input stream in bytes
\return -1 error
\return >=0 TODO
*/
DINT bgPVStructDeserializeJSON(char* pvNameRoot, char* fromStream, UDINT lengthStream);

#endif
```

### bgfsig.c
```c
#include <bur/plc.h>
#include <bur/plctypes.h>

#include "bglib/bgdebug.h"
#include "bglib/bgstring.h"
#include "bglib/bgSecMD5Signature.h"
#include "bgfsig.h"

/*define a limit for number of lines within a file*/
#define MAX_NUMBER_OF_LINES	3000

static int bgGetLineFromTextBuffer(char* pText, char** pLineNext, char* pDest, int maxLen, int* charCount);

#define  secretWord "NONE!"

/*=============================================================*/
int bgFileSignatureVerify(char *inFileBuffer, char *resultStringMinLen64)
{
int i, index;
char lineBuffer[255];
char lineBufferRaw[255];
int lineCount;
int charCount;
bgStringList_typ splitLine;
md5_state_t state;
md5_byte_t digest[16];
char hexDigestCalculated[40];
char hexDigestFromFile[40];

char *pLineCurrent;
char *pLineNext;

	/*init digest*/
	md5_init(&state);

	/*init hexDigestFromFile as empty*/
	hexDigestFromFile[0] = 0;

	/*init line ptr-s*/
	pLineCurrent = inFileBuffer;
	pLineNext = 0L;

	lineCount = 0;

	/*process all lines from the file*/
	while( 1 ){
	int isNextLinePresent;

		isNextLinePresent = bgGetLineFromTextBuffer(pLineCurrent, &pLineNext, lineBufferRaw, 255, &charCount);

		if( lineCount++ > MAX_NUMBER_OF_LINES){
			DBGCRT("Supplied file buffer has more then %d lines!\r\n", lineCount);
			if( resultStringMinLen64 )
				brsstrcpy((UDINT)resultStringMinLen64, (UDINT)"Err: file is too long!");
			return -2;
		}

		/*copy a trimmed line into the local buffer*/
		charCount = bgStrCpyNTrimLeadingSpaces(lineBuffer, lineBufferRaw, 255);

		/*check for empty lines & comments*/
		if( !charCount || (lineBuffer[0] == '*')){
			/*empty lines or comments -> skip and go to the next line*/
		}else{
			/*check if this is a signature line*/
			index = bgStrFind(lineBuffer, "SIGNATURE", -1, 0);
			if( index >= 0){
				/*line w. signature -> extract signature stored in the file*/
				splitLine.src = lineBuffer;
				bgStringSplitLine(&splitLine, '=');
				if( splitLine.itemCount != 2){
					DBGCRT("Can't extract signature from the supplied file buffer\r\n");
					if( resultStringMinLen64 )
						brsstrcpy((UDINT)resultStringMinLen64, (UDINT)"Err: can't extract signature");
					return -2;
				}
				/*copy extracted signature from the file into the local buffer*/
				bgStrCpyN(hexDigestFromFile, splitLine.items[1], 40);
				bgStringUpper(hexDigestFromFile);

			}else{
				/*line wo. signature -> use (append) for digest calculation*/
				md5_append(&state, (const md5_byte_t *)lineBuffer, strlen(lineBuffer));
			}
		}

		/*process next line*/
		if( isNextLinePresent )
			pLineCurrent = pLineNext;
		else
			break;
	}

	/*append secret content*/
	md5_append(&state, (const md5_byte_t *)secretWord, strlen(secretWord));

	/*generate digest*/
	md5_finish(&state, digest);

	/*convert calculated digest into a hex string*/
	for (i = 0; i < 16; ++i)
	    sprintf2(hexDigestCalculated + i * 2, "%02X", digest[i]);

	/*check if supplied file buffer had stored digital signature*/
	if( !hexDigestFromFile[0] ){
		/*digital signature was NOT present in this file->return result and current (calculated) file digest*/
		if( resultStringMinLen64 )
			sprintf2(resultStringMinLen64, "StoredSig=NONE CalcSig=%s\n\r", hexDigestCalculated);
		return 0;

	}else{
		/*digital signature IS present in this file->compare calculated and stored signaure*/

		for (i = 0; i < 32; i++){
			if(hexDigestCalculated[i] != hexDigestFromFile[i] ){
				/*digital signatures are not equal -> exit*/
				if( resultStringMinLen64 )
					sprintf2(resultStringMinLen64, "StoredSig=%s CalcSig=%s\n\r", hexDigestFromFile, hexDigestCalculated);

				return 2;
			}
		}

		/*digital signature verified! stored and calculated signatures are equal!*/
		if( resultStringMinLen64 )
			sprintf2(resultStringMinLen64, "StoredSigEQUALCalcSig=%s\n\r", hexDigestCalculated);

		return 1;

	}
}
/*=============================================================*/

/*
Input(s):
char *pText - ptr to the text buffer from which to extract a line
char *pDest - destination buffer where to copy the content of a line
int maxLen - max length of the destination buffer

Output(s):
char **pLineNext - ptr to the next line
int *charCount - total number of chars copied into the dest buffer

Return:
0 - there is no more lines in the supplied text buffer
1 - more lines are present in the supplied text buffer
*/
static int bgGetLineFromTextBuffer(char* pText, char** pLineNext, char* pDest, int maxLen, int* charCount)
{

unsigned char *ptrItemStart, *ptrItemEnd;
unsigned char *ptrCpyDest;

	/*init ptrs to the start of the text buffer*/
	ptrItemStart = pText;
	ptrItemEnd = pText;
	ptrCpyDest = pDest;

	/*basic check*/
	if( *ptrItemStart == 0){
		return 0;
	}

	*charCount = 0;
	while( 1 ){
		if( (*ptrItemEnd == 0x0D) || (*ptrItemEnd == 0x0A)){
			/*EOF line char found! -> exit*/
			ptrItemEnd++;

			/*check for an additional \r or \n*/
			if( (*ptrItemEnd == 0x0D) || (*ptrItemEnd == 0x0A)){
				ptrItemEnd++;
			}

			ptrItemStart = ptrItemEnd;

			/*terminate dest buffer*/
			*ptrCpyDest = 0;

			/*check for an end of the text*/
			if( (*ptrItemEnd == 0) ){
				*pLineNext = 0L;
				/*0 -> there are NO more lines in the text buffer*/
				return 0;
			}else{
				*pLineNext = ptrItemStart;
				/*1 -> there are more lines in the text buffer*/
				return 1;
			}
		}else
		if( *ptrItemEnd == 0){
			/*end of text buffer found! -> exit*/

			/*terminate dest buffer*/
			*ptrCpyDest = 0;

			*pLineNext = 0L;
			/*0 -> there are NO more lines in the text buffer*/
			return 0;
		}else{
			/*copy line content into the supplied dest buffer
			check for buffer overflow*/

			if( (*charCount) < maxLen ){
				*ptrCpyDest = *ptrItemEnd;
				ptrCpyDest++;
				(*charCount)++;
			}else{

				DBGCRT("Line is longer then the max allowed size!\r\n");

				/*terminate dest buffer*/
				*ptrCpyDest = 0;

				*pLineNext = 0L;
				/*0 -> there are NO more lines in the text buffer! Error*/
				return 0;
			}

			ptrItemEnd++;
		}
	}/*while*/
}
```

### bgSecMD5Signature.c
```c
#include "bgSecMD5Signature.h"
//#include <string.h>

#include <bur/plc.h>

/*
  Copyright (C) 2002 Aladdin Enterprises.  All rights reserved.

  Independent implementation of MD5 (RFC 1321).

  This code implements the MD5 Algorithm defined in RFC 1321, whose
  text is available at
	http://www.ietf.org/rfc/rfc1321.txt
  The code is derived from the text of the RFC, including the test suite
  (section A.5) but excluding the rest of Appendix A.  It does not include
  any code or documentation that is identified in the RFC as being
  copyrighted.

  The original and principal author of md5.c is L. Peter Deutsch
  <ghost@aladdin.com>.  Other authors are noted in the change history
  that follows (in reverse chronological order):

  2002-04-13 lpd Splits off main program into a separate file, md5main.c.
 */

#undef BYTE_ORDER	/* 1 = big-endian, -1 = little-endian, 0 = unknown */
#ifdef ARCH_IS_BIG_ENDIAN
#define BYTE_ORDER (ARCH_IS_BIG_ENDIAN ? 1 : -1)
#else
#define BYTE_ORDER 0
#endif

#define T_MASK ((md5_word_t)~0)
#define T1 /* 0xd76aa478 */ (T_MASK ^ 0x28955b87)
#define T2 /* 0xe8c7b756 */ (T_MASK ^ 0x173848a9)
#define T3    0x242070db
#define T4 /* 0xc1bdceee */ (T_MASK ^ 0x3e423111)
#define T5 /* 0xf57c0faf */ (T_MASK ^ 0x0a83f050)
#define T6    0x4787c62a
#define T7 /* 0xa8304613 */ (T_MASK ^ 0x57cfb9ec)
#define T8 /* 0xfd469501 */ (T_MASK ^ 0x02b96afe)
#define T9    0x698098d8
#define T10 /* 0x8b44f7af */ (T_MASK ^ 0x74bb0850)
#define T11 /* 0xffff5bb1 */ (T_MASK ^ 0x0000a44e)
#define T12 /* 0x895cd7be */ (T_MASK ^ 0x76a32841)
#define T13    0x6b901122
#define T14 /* 0xfd987193 */ (T_MASK ^ 0x02678e6c)
#define T15 /* 0xa679438e */ (T_MASK ^ 0x5986bc71)
#define T16    0x49b40821
#define T17 /* 0xf61e2562 */ (T_MASK ^ 0x09e1da9d)
#define T18 /* 0xc040b340 */ (T_MASK ^ 0x3fbf4cbf)
#define T19    0x265e5a51
#define T20 /* 0xe9b6c7aa */ (T_MASK ^ 0x16493855)
#define T21 /* 0xd62f105d */ (T_MASK ^ 0x29d0efa2)
#define T22    0x02441453
#define T23 /* 0xd8a1e681 */ (T_MASK ^ 0x275e197e)
#define T24 /* 0xe7d3fbc8 */ (T_MASK ^ 0x182c0437)
#define T25    0x21e1cde6
#define T26 /* 0xc33707d6 */ (T_MASK ^ 0x3cc8f829)
#define T27 /* 0xf4d50d87 */ (T_MASK ^ 0x0b2af278)
#define T28    0x455a14ed
#define T29 /* 0xa9e3e905 */ (T_MASK ^ 0x561c16fa)
#define T30 /* 0xfcefa3f8 */ (T_MASK ^ 0x03105c07)
#define T31    0x676f02d9
#define T32 /* 0x8d2a4c8a */ (T_MASK ^ 0x72d5b375)
#define T33 /* 0xfffa3942 */ (T_MASK ^ 0x0005c6bd)
#define T34 /* 0x8771f681 */ (T_MASK ^ 0x788e097e)
#define T35    0x6d9d6122
#define T36 /* 0xfde5380c */ (T_MASK ^ 0x021ac7f3)
#define T37 /* 0xa4beea44 */ (T_MASK ^ 0x5b4115bb)
#define T38    0x4bdecfa9
#define T39 /* 0xf6bb4b60 */ (T_MASK ^ 0x0944b49f)
#define T40 /* 0xbebfbc70 */ (T_MASK ^ 0x4140438f)
#define T41    0x289b7ec6
#define T42 /* 0xeaa127fa */ (T_MASK ^ 0x155ed805)
#define T43 /* 0xd4ef3085 */ (T_MASK ^ 0x2b10cf7a)
#define T44    0x04881d05
#define T45 /* 0xd9d4d039 */ (T_MASK ^ 0x262b2fc6)
#define T46 /* 0xe6db99e5 */ (T_MASK ^ 0x1924661a)
#define T47    0x1fa27cf8
#define T48 /* 0xc4ac5665 */ (T_MASK ^ 0x3b53a99a)
#define T49 /* 0xf4292244 */ (T_MASK ^ 0x0bd6ddbb)
#define T50    0x432aff97
#define T51 /* 0xab9423a7 */ (T_MASK ^ 0x546bdc58)
#define T52 /* 0xfc93a039 */ (T_MASK ^ 0x036c5fc6)
#define T53    0x655b59c3
#define T54 /* 0x8f0ccc92 */ (T_MASK ^ 0x70f3336d)
#define T55 /* 0xffeff47d */ (T_MASK ^ 0x00100b82)
#define T56 /* 0x85845dd1 */ (T_MASK ^ 0x7a7ba22e)
#define T57    0x6fa87e4f
#define T58 /* 0xfe2ce6e0 */ (T_MASK ^ 0x01d3191f)
#define T59 /* 0xa3014314 */ (T_MASK ^ 0x5cfebceb)
#define T60    0x4e0811a1
#define T61 /* 0xf7537e82 */ (T_MASK ^ 0x08ac817d)
#define T62 /* 0xbd3af235 */ (T_MASK ^ 0x42c50dca)
#define T63    0x2ad7d2bb
#define T64 /* 0xeb86d391 */ (T_MASK ^ 0x14792c6e)

static void
md5_process(md5_state_t *pms, const md5_byte_t *data /*[64]*/)
{
    md5_word_t
	a = pms->abcd[0], b = pms->abcd[1],
	c = pms->abcd[2], d = pms->abcd[3];
    md5_word_t t;
#if BYTE_ORDER > 0
    /* Define storage only for big-endian CPUs. */
    md5_word_t X[16];
#else
    /* Define storage for little-endian or both types of CPUs. */
    md5_word_t xbuf[16];
    const md5_word_t *X;
#endif

    {
#if BYTE_ORDER == 0
	/*
	 * Determine dynamically whether this is a big-endian or
	 * little-endian machine, since we can use a more efficient
	 * algorithm on the latter.
	 */
	static const int w = 1;

	if (*((const md5_byte_t *)&w)) /* dynamic little-endian */
#endif
#if BYTE_ORDER <= 0		/* little-endian */
	{
	    /*
	     * On little-endian machines, we can process properly aligned
	     * data without copying it.
	     */
	    if (!((data - (const md5_byte_t *)0) & 3)) {
		/* data are properly aligned */
		X = (const md5_word_t *)data;
	    } else {
		/* not aligned */
		memcpy(xbuf, data, 64);
		X = xbuf;
	    }
	}
#endif
#if BYTE_ORDER == 0
	else			/* dynamic big-endian */
#endif
#if BYTE_ORDER >= 0		/* big-endian */
	{
	    /*
	     * On big-endian machines, we must arrange the bytes in the
	     * right order.
	     */
	    const md5_byte_t *xp = data;
	    int i;

#if BYTE_ORDER == 0
	    X = xbuf;		/* (dynamic only) */
#else
#define xbuf X		/* (static only) */
#endif
	    for (i = 0; i < 16; ++i, xp += 4)
		xbuf[i] = xp[0] + (xp[1] << 8) + (xp[2] << 16) + (xp[3] << 24);
	}
#endif
    }

#define ROTATE_LEFT(x, n) (((x) << (n)) | ((x) >> (32 - (n))))

    /* Round 1. */
    /* Let [abcd k s i] denote the operation
       a = b + ((a + F(b,c,d) + X[k] + T[i]) <<< s). */
#define F(x, y, z) (((x) & (y)) | (~(x) & (z)))
#define SET(a, b, c, d, k, s, Ti)\
  t = a + F(b,c,d) + X[k] + Ti;\
  a = ROTATE_LEFT(t, s) + b
    /* Do the following 16 operations. */
    SET(a, b, c, d,  0,  7,  T1);
    SET(d, a, b, c,  1, 12,  T2);
    SET(c, d, a, b,  2, 17,  T3);
    SET(b, c, d, a,  3, 22,  T4);
    SET(a, b, c, d,  4,  7,  T5);
    SET(d, a, b, c,  5, 12,  T6);
    SET(c, d, a, b,  6, 17,  T7);
    SET(b, c, d, a,  7, 22,  T8);
    SET(a, b, c, d,  8,  7,  T9);
    SET(d, a, b, c,  9, 12, T10);
    SET(c, d, a, b, 10, 17, T11);
    SET(b, c, d, a, 11, 22, T12);
    SET(a, b, c, d, 12,  7, T13);
    SET(d, a, b, c, 13, 12, T14);
    SET(c, d, a, b, 14, 17, T15);
    SET(b, c, d, a, 15, 22, T16);
#undef SET

     /* Round 2. */
     /* Let [abcd k s i] denote the operation
          a = b + ((a + G(b,c,d) + X[k] + T[i]) <<< s). */
#define G(x, y, z) (((x) & (z)) | ((y) & ~(z)))
#define SET(a, b, c, d, k, s, Ti)\
  t = a + G(b,c,d) + X[k] + Ti;\
  a = ROTATE_LEFT(t, s) + b
     /* Do the following 16 operations. */
    SET(a, b, c, d,  1,  5, T17);
    SET(d, a, b, c,  6,  9, T18);
    SET(c, d, a, b, 11, 14, T19);
    SET(b, c, d, a,  0, 20, T20);
    SET(a, b, c, d,  5,  5, T21);
    SET(d, a, b, c, 10,  9, T22);
    SET(c, d, a, b, 15, 14, T23);
    SET(b, c, d, a,  4, 20, T24);
    SET(a, b, c, d,  9,  5, T25);
    SET(d, a, b, c, 14,  9, T26);
    SET(c, d, a, b,  3, 14, T27);
    SET(b, c, d, a,  8, 20, T28);
    SET(a, b, c, d, 13,  5, T29);
    SET(d, a, b, c,  2,  9, T30);
    SET(c, d, a, b,  7, 14, T31);
    SET(b, c, d, a, 12, 20, T32);
#undef SET

     /* Round 3. */
     /* Let [abcd k s t] denote the operation
          a = b + ((a + H(b,c,d) + X[k] + T[i]) <<< s). */
#define H(x, y, z) ((x) ^ (y) ^ (z))
#define SET(a, b, c, d, k, s, Ti)\
  t = a + H(b,c,d) + X[k] + Ti;\
  a = ROTATE_LEFT(t, s) + b
     /* Do the following 16 operations. */
    SET(a, b, c, d,  5,  4, T33);
    SET(d, a, b, c,  8, 11, T34);
    SET(c, d, a, b, 11, 16, T35);
    SET(b, c, d, a, 14, 23, T36);
    SET(a, b, c, d,  1,  4, T37);
    SET(d, a, b, c,  4, 11, T38);
    SET(c, d, a, b,  7, 16, T39);
    SET(b, c, d, a, 10, 23, T40);
    SET(a, b, c, d, 13,  4, T41);
    SET(d, a, b, c,  0, 11, T42);
    SET(c, d, a, b,  3, 16, T43);
    SET(b, c, d, a,  6, 23, T44);
    SET(a, b, c, d,  9,  4, T45);
    SET(d, a, b, c, 12, 11, T46);
    SET(c, d, a, b, 15, 16, T47);
    SET(b, c, d, a,  2, 23, T48);
#undef SET

     /* Round 4. */
     /* Let [abcd k s t] denote the operation
          a = b + ((a + I(b,c,d) + X[k] + T[i]) <<< s). */
#define I(x, y, z) ((y) ^ ((x) | ~(z)))
#define SET(a, b, c, d, k, s, Ti)\
  t = a + I(b,c,d) + X[k] + Ti;\
  a = ROTATE_LEFT(t, s) + b
     /* Do the following 16 operations. */
    SET(a, b, c, d,  0,  6, T49);
    SET(d, a, b, c,  7, 10, T50);
    SET(c, d, a, b, 14, 15, T51);
    SET(b, c, d, a,  5, 21, T52);
    SET(a, b, c, d, 12,  6, T53);
    SET(d, a, b, c,  3, 10, T54);
    SET(c, d, a, b, 10, 15, T55);
    SET(b, c, d, a,  1, 21, T56);
    SET(a, b, c, d,  8,  6, T57);
    SET(d, a, b, c, 15, 10, T58);
    SET(c, d, a, b,  6, 15, T59);
    SET(b, c, d, a, 13, 21, T60);
    SET(a, b, c, d,  4,  6, T61);
    SET(d, a, b, c, 11, 10, T62);
    SET(c, d, a, b,  2, 15, T63);
    SET(b, c, d, a,  9, 21, T64);
#undef SET

     /* Then perform the following additions. (That is increment each
        of the four registers by the value it had before this block
        was started.) */
    pms->abcd[0] += a;
    pms->abcd[1] += b;
    pms->abcd[2] += c;
    pms->abcd[3] += d;
}

void
md5_init(md5_state_t *pms)
{
    pms->count[0] = pms->count[1] = 0;
    pms->abcd[0] = 0x67452301;
    pms->abcd[1] = /*0xefcdab89*/ T_MASK ^ 0x10325476;
    pms->abcd[2] = /*0x98badcfe*/ T_MASK ^ 0x67452301;
    pms->abcd[3] = 0x10325476;
}

void
md5_append(md5_state_t *pms, const md5_byte_t *data, int nbytes)
{
    const md5_byte_t *p = data;
    int left = nbytes;
    int offset = (pms->count[0] >> 3) & 63;
    md5_word_t nbits = (md5_word_t)(nbytes << 3);

    if (nbytes <= 0)
	return;

    /* Update the message length. */
    pms->count[1] += nbytes >> 29;
    pms->count[0] += nbits;
    if (pms->count[0] < nbits)
	pms->count[1]++;

    /* Process an initial partial block. */
    if (offset) {
	int copy = (offset + nbytes > 64 ? 64 - offset : nbytes);

	memcpy(pms->buf + offset, p, copy);
	if (offset + copy < 64)
	    return;
	p += copy;
	left -= copy;
	md5_process(pms, pms->buf);
    }

    /* Process full blocks. */
    for (; left >= 64; p += 64, left -= 64)
	md5_process(pms, p);

    /* Process a final partial block. */
    if (left)
	memcpy(pms->buf, p, left);
}

void
md5_finish(md5_state_t *pms, md5_byte_t digest[16])
{
    static const md5_byte_t pad[64] = {
	0x80, 0, 0, 0, 0, 0, 0, 0, 0, 0, 0, 0, 0, 0, 0, 0,
	0, 0, 0, 0, 0, 0, 0, 0, 0, 0, 0, 0, 0, 0, 0, 0,
	0, 0, 0, 0, 0, 0, 0, 0, 0, 0, 0, 0, 0, 0, 0, 0,
	0, 0, 0, 0, 0, 0, 0, 0, 0, 0, 0, 0, 0, 0, 0, 0
    };
    md5_byte_t data[8];
    int i;

    /* Save the length before padding. */
    for (i = 0; i < 8; ++i)
	data[i] = (md5_byte_t)(pms->count[i >> 2] >> ((i & 3) << 3));
    /* Pad to 56 bytes mod 64. */
    md5_append(pms, pad, ((55 - (pms->count[0] >> 3)) & 63) + 1);
    /* Append the length. */
    md5_append(pms, data, 8);
    for (i = 0; i < 16; ++i)
	digest[i] = (md5_byte_t)(pms->abcd[i >> 2] >> ((i & 3) << 3));
}

int
md5_selftest(void)
{
    static const char *const test[7*2] = {
	"", "d41d8cd98f00b204e9800998ecf8427e",
	"a", "0cc175b9c0f1b6a831c399e269772661",
	"abc", "900150983cd24fb0d6963f7d28e17f72",
	"message digest", "f96b697d7cb7938d525a2f31aaf161d0",
	"abcdefghijklmnopqrstuvwxyz", "c3fcd3d76192e4007dfb496cca67e13b",
	"ABCDEFGHIJKLMNOPQRSTUVWXYZabcdefghijklmnopqrstuvwxyz0123456789",
				"d174ab98d277d9f5a5611c2c9f419d9f",
	"12345678901234567890123456789012345678901234567890123456789012345678901234567890", "57edf4a22be3c955ac49da2e2107b67a"
    };
    int i;
    int status = 0;

    for (i = 0; i < 7*2; i += 2) {
	md5_state_t state;
	md5_byte_t digest[16];
	char hex_output[16*2 + 1];
	int di;

	md5_init(&state);
	md5_append(&state, (const md5_byte_t *)test[i], strlen(test[i]));
	md5_finish(&state, digest);
	for (di = 0; di < 16; ++di)
	    bgsprintf(hex_output + di * 2, "%02x", digest[di]);
	if (strcmp(hex_output, test[i + 1])) {
#if 0
	    printf("MD5 (\"%s\") = ", test[i]);
	    puts(hex_output);
	    printf("**** ERROR, should be: %s\n", test[i + 1]);
#endif
	    status = 1;
	}
    }
    if (status == 0);

#if 0
		puts("md5 self-test completed successfully.");
#endif

    return status;
}
```

### Package Logical/paiComponents/paiHmi - pai HMI related components

### paiHmiMsgRunning.typ
```iecst
(********************************************************************
 * COPYRIGHT -- pai
 ********************************************************************
 * Package: HMI
 * File: HMI.typ
 * Author: goran
 * Created: August 28, 2015
 ********************************************************************
 * Data types of package HMI
 ********************************************************************)
(*########################################################################*)
(*HMI object - Running Messages (i.e. content scrolls )*)
(*########################################################################*)

TYPE
	paiHmiMsgRunning_typ : 	STRUCT  (*0-disable; 1-enable*)
		iEnable : BOOL; (*input: address of the alarm array*)
		iScrollMode : UDINT; (*scroll mode*)
		iScrollLength : UDINT; (*scroll length*)
		iScrollDelayXms : UDINT; (*scroll speed*)
		iMsgAddr : UDINT; (*address of the message for scroll*)
		oMsg : STRING[255]; (*output: message ID of the active alarm / message*)
		oMsgVisible : UINT; (*output: visibilty control DP for the VC text message*)
		oMsgFCIdx : UINT; (*output: visibilty control DP for the VC text message*)
		state : UINT; (*Status for common dialog layer*)
		curIdx : UINT; (*Status for common dialog layer*)
		tmr1 : TON; (*Dialog control timer*)
	END_STRUCT;
END_TYPE
```

### paiHmiSystemNetworking.typ
```iecst
(********************************************************************
 * COPYRIGHT -- pai
 ********************************************************************
 * Package: paiHMI
 * File: paiHmiSystemNetworking.typ
 * Author: goran
 * Created: August 28, 2013
 *********************************************************************)
(*########################################################################*)
(*HMI object - System Time*)
(*########################################################################*)

TYPE
	paiHmiNumericalNetworkAddr_typ : 	STRUCT
		ipAddr : ARRAY[0..3]OF USINT;
		netMask : ARRAY[0..3]OF USINT;
		broadcast : ARRAY[0..3]OF USINT;
		gateway : ARRAY[0..3]OF USINT;
	END_STRUCT;
	paiHmiSystemNetworking_typ : 	STRUCT
		iChangeNWSettings : BOOL;
		iConfigIsValid : BOOL;
		iPtrNWConfig : REFERENCE TO paiARNetworkAddress_typ;
		oCurrentNWSettings : paiARNetworkAddress_typ;
		oNumericalNWSettings : paiHmiNumericalNetworkAddr_typ;
		oError : UDINT;
		oErrorText : STRING[63];
		oState : UDINT;
		mGetIpAddr : CfgGetIPAddr;
		mSetIpAddr : CfgSetIPAddr;
		mGetSubnetMask : CfgGetSubnetMask;
		mSetSubnetMask : CfgSetSubnetMask;
		mGetBroadcastAddr : CfgGetBroadcastAddr;
		mSetBroadcastAddr : CfgSetBroadcastAddr;
		mGetDefaultGateway : CfgGetDefaultGateway;
		mSetDefaultGateway : CfgSetDefaultGateway;
		mGetHostName : CfgGetHostName;
		mSetHostHame : CfgSetHostName;
		New_Member1 : USINT;
		New_Member : USINT;
		New_Member2 : USINT;
	END_STRUCT;
END_TYPE
```

### paiHmiTemplate.typ
```iecst
(********************************************************************
 * COPYRIGHT --
 ********************************************************************
 * Package: HMI
 * File: cfgPaiHmiTemplate.typ
 * Author: goran
 * Created: October 15, 2014
 ********************************************************************
 * Data types of package HMI
 ********************************************************************)
(*########################################################################*)
(*HMI key assinged PV-s (i.e. page navigation, save btns, etc)*)
(*########################################################################*)
(*########################################################################*)
(*HMI key assinged PV-s (i.e. menu, tabs, etc)*)
(*########################################################################*)

TYPE
	paiHmiTemplateKeys_typ : 	STRUCT
		menuKeyTopLT : INT; (*Menu key press top LF*)
		menuKeyTopRT : INT; (*Mom keys connected to menu items RT*)
		currentMenuLF : INT;
		currentMenuRT : INT;
		tabKeysRadioDataPoint : INT; (*DP that tab button are writing to in order to create radio buttons/tab view effect*)
		tabKeysRadioDataPointOld : INT; (*DP that tab button are writing to in order to create radio buttons/tab view effect*)
		tabKeysRadioArray : ARRAY[0..paiHMI_ENUM_TABS_MAXIDX]OF INT;
	END_STRUCT;
END_TYPE

(*########################################################################*)
(*HMI related status control PV-s (i.e. visibility, locking, etc)*)
(*########################################################################*)

TYPE
	paiHmiTemplateStatus_typ : 	STRUCT
		menuVisibleLT : UINT; (*Main menu LF visibility control *)
		menuIndexLT : UINT; (*Main menu currently selected menu item - LF*)
		loginVisibleGE1 : USINT; (*Visibility control for login level related stuff - set to visible (0) if login level >= 1; othervise set to 1 (i.e. loginLevel < 1)*)
		loginVisibleGE2 : USINT; (*Visibility control for login level related stuff - set to visible (0) if login level >= 2; othervise set to 1 (i.e. loginLevel < 2)*)
		menuLFHideTimer : TON; (*timer of automaticaly hiding LF dropdown menu*)
		unusedItemInvisible : UDINT; (*used for VC items that are not used (hidden)*)
		passwordStrings : ARRAY[0..paiHMI_PWD_LEVELS]OF STRING[paiHMI_PWD_MAXLEN]; (*Password strings used for loginLevel control*)
	END_STRUCT;
END_TYPE

(*########################################################################*)
(*HMI related timer settings*)
(*########################################################################*)

TYPE
	paiHmiTemplateTimerSettings_typ : 	STRUCT
		loginTimeout : REAL; (*Login timeout timer setting*)
		dialogBoxTimeout : REAL; (*Dialog box (i.e. save data? yes/no) timeout for waiting on input*)
		splashScreenTimeout : REAL; (*Duration of the initial screen (i.e. manufacturer logo) *)
		dropdwMenuLFTimeout : REAL; (*Duration after which a dropdown menu is automaticaly hiden if not clicked *)
	END_STRUCT;
END_TYPE

(*########################################################################*)
(*HMI pwd settings*)
(*########################################################################*)

TYPE
	paiHmiTemplatePwdSettings_typ : 	STRUCT
		passwordAdmin : STRING[paiHMI_PWD_MAXLEN]; (*Login timeout timer setting*)
		passwordMaint : STRING[paiHMI_PWD_MAXLEN]; (*Login timeout timer setting*)
		passwordSupervisor : STRING[paiHMI_PWD_MAXLEN]; (*Login timeout timer setting*)
		passwordFactory : STRING[paiHMI_PWD_MAXLEN]; (*Login timeout timer setting*)
	END_STRUCT;
END_TYPE

(*########################################################################*)
(*HMI related PV-s connected to VC runtime (see VC runtime settings)*)
(*########################################################################*)

TYPE
	paiHmiTemplateVCRuntime_typ : 	STRUCT
		wheelCount : INT;
		wheelEnter : INT;
		keyLevelChange : INT;
		keyLevelCurrent : INT;
		languageChange : INT;
		languageCurrent : INT;
		keyMatrix : ARRAY[0..63]OF INT;
		LEDMatrix : ARRAY[0..63]OF INT;
		pageChange : INT;
		pageCurrent : INT;
		lifeSign : INT;
		IPAddress : STRING[31];
		focusControl : INT;
		helpControl : INT;
		touchCalibration : INT;
		touchCalibrationState : INT;
		screenSaverTimeout_sec : INT;
		screenSaverPage : INT;
	END_STRUCT;
END_TYPE

(*########################################################################*)
(*HMI related config file settings*)
(*########################################################################*)

TYPE
	paiHmiTemplateConfig_typ : 	STRUCT
		pwdSettings : paiHmiTemplatePwdSettings_typ;
		timerSettings : paiHmiTemplateTimerSettings_typ;
	END_STRUCT;
END_TYPE

(*########################################################################*)
(*HMI control logic private PV-s*)
(*########################################################################*)

TYPE
	paiHmiTemplateItem_typ : 	STRUCT
		itemText : STRING[31];
		itemVisible : UINT;
		itemDisabled : UINT;
		jumpPageId : UINT;
	END_STRUCT;
	paiHmiTemplateSubmenuItem_typ : 	STRUCT
		button : paiHmiTemplateItem_typ;
		tabs : ARRAY[0..paiHMI_ENUM_TABS_MAXIDX]OF paiHmiTemplateItem_typ;
	END_STRUCT;
	paiHmiTemplatePrivate_typ : 	STRUCT
		initDone : BOOL;
		state : INT;
		vcHandle : UDINT;
		index : UDINT;
		indexButton : UDINT;
		indexTab : UDINT;
		TG_id : UDINT;
		text : STRING[paiHMI_ENUM_TG_TEXT_MAXLEN];
		parseErrorText : STRING[127];
		textLen : UINT;
		textLines : ARRAY[0..paiHMI_ENUM_TG_TEXT_MAXIDX]OF STRING[paiHMI_ENUM_TG_TEXT_MAXLEN];
		activeTabs : ARRAY[0..paiHMI_ENUM_TABS_MAXIDX]OF paiHmiTemplateItem_typ;
		menuLF : ARRAY[0..paiHMI_ENUM_MENU_ITEMS_LT]OF paiHmiTemplateSubmenuItem_typ;
		pageSetByLFMenu : INT;
		pageCurrent : UDINT;
		pagePrev : UDINT;
		pageInit : BOOL;
		pageExit : BOOL;
	END_STRUCT;
	paiHmiTemplate_typ : 	STRUCT
		runtime : paiHmiTemplateVCRuntime_typ; (*VC runtime Datapoint PV-s. Assigned to different VC control points.*)
		status : paiHmiTemplateStatus_typ;
		keys : paiHmiTemplateKeys_typ;
		timerSettings : paiHmiTemplateTimerSettings_typ;
		activeTabs : ARRAY[0..paiHMI_ENUM_TABS_MAXIDX]OF paiHmiTemplateItem_typ;
		activeTopMenuLF : paiHmiTemplateItem_typ;
		currentMenuLF : INT;
		currentTab : INT;
		prv : paiHmiTemplatePrivate_typ;
	END_STRUCT;
END_TYPE
```

### paiHmiParamList.c
```c
/********************************************************************
 * COPYRIGHT -- pai
 ********************************************************************
 * Program: hmilogic
 * File: hmiParamList.c
 * Author: goran
 * Created: September 05, 2013
 *******************************************************************/

#include <bur/plctypes.h>
#ifdef _DEFAULT_INCLUDES
	#include <AsDefault.h>
#endif

#define HMI_PARAMLIST_DECPLACES_DEFAULT  2 //default value of decimal places for any real number converted to text. Application specific.

/**
Bit manipulaiton utility functions.
 */
//#include <../../bglib/bgBitUtilities.h>

/**
String manipulaiton utility functions.
 */
//#include "../../paiComponents/bglib/bgsprintf.h"
#include "../../paiComponents/bglib/bgstring.h"
#include "../../paiComponents/Libraries/sprintf2/sprintf2.h"

/**
 Timer control utility functions.
 */
//#include <../../bglib/bgTimer1ms.h>

/*
###############################################################################
HMI table editor support. Set of functions that support table based editing of the parametars.
###############################################################################
*/

/**
rouding of a floating point value to the number of required decimal positions.
\param d value
\param pp number of decimal places
\return rounded value

*/
static float roundVal(float d, int ppOffset)
{

	int valInt;
	float exp10topp = 10.0;
	int count = 0;
	int pp = ppOffset;

	if(!pp){
		exp10topp = 1.0;
	}else
		if(pp<0){
		exp10topp = 0.1;
		count = (0 - pp) - 1;
	}else{
		exp10topp = 10.0;
		count = pp - 1;
	}

	while(count--){
		exp10topp *= exp10topp;
	}

	valInt = (int) (d *  exp10topp + 0.5);
	return ( valInt  /  exp10topp  );
}

/**
ftoa (float to ascii converion) with the added support for required number of decimal places in the text ouput.
\param value value to convert
\param pp number of decimal places
\return rounded value

*/
static void ftoaEx(float value, char* pText, int decPlacesOffset)
{
	char text[32];

	int len;
	int comaPos;
	int apendZerosCount;
	int ii;
	float rnd_val;
	int decPlaces = HMI_PARAMLIST_DECPLACES_DEFAULT + decPlacesOffset;

	if(!pText)
		return;

	//limit max dec places
	if(decPlaces > 5)
		decPlaces = 5;

	//convert float to ascii
	//	ftoa(value, text);
	rnd_val = roundVal(value, decPlaces);
	ftoa(rnd_val , (UDINT)text);

	//get the length of the converted string
	len = brsstrlen((UDINT)text);
	if(!len){
		//0 length > don't know what to do
		brsstrcpy((UDINT)pText, (UDINT)"?");
		return;
	}

	//find position of the coma
	comaPos = bgStrFind(text, ".", -1, -1);

	if(!decPlaces){
		//dec places are not needed

		if(comaPos>0){
			//coma is present > terminate the string at the comma position
			text[comaPos] = 0;
		}

	}else{
		//dec places are needed

		if(comaPos<0){
			//no coma present but it is needed
			brsstrcat((UDINT)text, (UDINT)".");
			len+=1;
			comaPos=len-1;
		}

		apendZerosCount = decPlaces - (len - comaPos - 1);

		if(apendZerosCount < 0){
			//too many digits after a decimal place > terminate string to a specified number of dec places
			apendZerosCount = 0 - apendZerosCount;
			text[len - apendZerosCount]=0;
		}else{
			//need to add zeros to satisfy the number of dec places
			for(ii=0; ii<apendZerosCount; ii++){
				text[len+ii]='0';
			}
			text[len+ii]=0;
		}
	}

	brsstrcpy((UDINT)pText, (UDINT)text);
	return;
}

static float hmiParamListTableGetPLCValue(UDINT pValue, REAL k_factor, REAL n_factor, int valueType)
{
	UDINT* pUdint = (UDINT*)pValue;
	float* pFloat = (float*)pValue;
	REAL tempReal;

	switch(valueType){
		case 1:
			if(pFloat){
				tempReal = ((float)(*pFloat)) * k_factor + n_factor;
			}else{
				tempReal = 0.0;
			}
			break;
		default:
			if(pUdint){
				tempReal = ((float)(*pUdint)) * k_factor + n_factor;
			}else{
				tempReal = 0.0;
			}
			break;
	}

	return tempReal;
}

static void hmiParamListTableDisplayToValue(float value, UDINT pValue, char* pOutputText,  int decPlaces, REAL k_factor, REAL n_factor, int valueType)
{
/*
scaling
y=kx + n
y=display value
x=plc value

x = (y- n)*(1/k)

value types:
0-UDINT
1-REAL

*/

	UDINT* pUdint = (UDINT*)pValue;
	float *pFloat = (float*)pValue;

	if(!k_factor){
		brsstrcpy((UDINT)pOutputText, (UDINT)"ERR: div by 0");
		return;
	}

	switch(valueType){
		case 1:
			*pFloat = (float)((value - n_factor) / k_factor);
			break;
		default:
			*pUdint = (UDINT)((value - n_factor) / k_factor);
			break;
	}

	ftoaEx(value, pOutputText, decPlaces);
}

static void hmiParamListTableValueToDisplay(UDINT pValue, char* pOutputText, float* pOutputFloat, int decPlaces, REAL k_factor, REAL n_factor, int valueType)
{
/*
scaling
y=kx + n
y=display value
x=plc value
*/
	REAL tempReal = hmiParamListTableGetPLCValue(pValue, k_factor, n_factor, valueType);

	if(pOutputFloat)
		*pOutputFloat = tempReal;

	ftoaEx(tempReal, pOutputText, decPlaces);
}

 void hmiParamListTableAddEntryNext(hmiParamListTable_typ* p, UDINT pValue, char* pName,
REAL valDefault, REAL valMin, REAL valMax, int decPlaces, REAL k_factor, REAL n_factor, UINT valueType, char* pDescription)
{
	if(!p)
		return;

	if(p->index >= hmiTableMAXENTRIES){
		brsstrcpy((UDINT)p->listValueText[p->index], (UDINT)"table overflow!");
		return;
	}

	p->listValuePtr[p->index] = pValue;
	sprintf2(p->listIdText[p->index], "%d", p->index);
	if(pDescription){
		bgStrCpyN(p->listDescription[p->index], pDescription, sizeof(p->listDescription[0]));
	}else{
		bgStrCpyN(p->listDescription[p->index], "no description", sizeof(p->listDescription[0]));
	}
	if(pName){
		bgStrCpyN(p->listName[p->index], pName, sizeof(p->listName[0]));
	}else{
		bgStrCpyN(p->listName[p->index], "no name", sizeof(p->listName[0]));
	}
	p->listDecPlaces[p->index] = decPlaces;

	p->listLimits[p->index].defaultValue = valDefault;
	p->listLimits[p->index].minValue= valMin;
	p->listLimits[p->index].maxValue= valMax;
	p->listLimits[p->index].k_factor= k_factor;
	p->listLimits[p->index].n_factor= n_factor;
	p->listLimits[p->index].valueType= valueType;

	hmiParamListTableValueToDisplay(p->listValuePtr[p->index],
		p->listValueText[p->index], 0, p->listDecPlaces[p->index], p->listLimits[p->index].k_factor, p->listLimits[p->index].n_factor, p->listLimits[p->index].valueType);

	p->index++;
	p->maxIndex++;
}

void hmiParamListTableEntryFirst(hmiParamListTable_typ* p, char* pListName)
{
	int ii;

	p->maxIndex = 0;
	p->index = 0;
	bgStrCpyN(p->listHeader, pListName, sizeof(p->listHeader));

	//clear all names from the list
	for(ii=0; ii<=hmiTableMAXENTRIES;ii++){
		brsstrcpy((UDINT)p->listIdText[ii], (UDINT)"");
		brsstrcpy((UDINT)p->listName[ii], (UDINT)"");
		brsstrcpy((UDINT)p->listValueText[ii], (UDINT)"");
	}
}

void hmiParamListTableEntryLast(hmiParamListTable_typ* p)
{
	if(p->maxIndex)
		p->maxIndex--;

	//init index value
	p->index = 0;

	//update text fields according to the currently selected table element
	bgStrCpyN(p->selName, p->listName[p->index], sizeof(p->selName));
	bgStrCpyN(p->selDescription, p->listDescription[p->index], sizeof(p->selDescription));

	//set limits on the HMI input control that coresponds to the currently selected table element
	p->selValueREALMin = p->listLimits[p->index].minValue;
	p->selValueREALMax= p->listLimits[p->index].maxValue;
	p->selValueREALDefault = p->listLimits[p->index].defaultValue;
	p->selValueDecPlaces = p->listDecPlaces[p->index];

	//display selected table element
	hmiParamListTableValueToDisplay(p->listValuePtr[p->index],
		p->listValueText[p->index], &p->selValueREAL, p->listDecPlaces[p->index], p->listLimits[p->index].k_factor, p->listLimits[p->index].n_factor, p->listLimits[p->index].valueType);

}

//
//void hmiParamListTableCyclic(hmiParamListTable_typ* p)
//{
//	if(!p)
//		return;
//
//	//limit index to max index value (up arrow)
//	if(p->index >= p->maxIndex){
//		p->index = p->maxIndex;
//	}
//
//	//keep checking if index changes (i.e. user changes entry selection)
//	if(p->index != p->indexOld){
//		//index change > update selected value for user entry
//		p->indexOld = p->index;
//		hmiParamListTableValueToDisplay(p->listValuePtr[p->index], p->listValueText[p->index],
//			&p->selValueREAL, p->listDecPlaces[p->index], p->listLimits[p->index].k_factor, p->listLimits[p->index].n_factor, p->listLimits[p->index].valueType);
//		//store value for change detection
//		p->selValueREALOld = p->selValueREAL;
//
//		//update text fields
//		bgStrCpyN(p->selName, p->listName[p->index], sizeof(p->selName));
//		bgStrCpyN(p->selDescription, p->listDescription[p->index], sizeof(p->selDescription));
//
//		//set limits for the selected element
//		p->selValueREALMin = p->listLimits[p->index].minValue;
//		p->selValueREALMax= p->listLimits[p->index].maxValue;
//		p->selValueREALDefault = p->listLimits[p->index].defaultValue;
//		p->selValueDecPlaces = p->listDecPlaces[p->index];
//
//	}
//
//
//	//keep checking if currently selected value changes(i.e. user enteres new value)
//	if(p->selValueREALOld != p->selValueREAL){
//		if(p->selValueREALMin < p->selValueREALMax){
//			//enforce limits
//			if(p->selValueREAL < p->selValueREALMin)
//				p->selValueREAL = p->selValueREALMin;
//
//			if(p->selValueREAL > p->selValueREALMax)
//				p->selValueREAL = p->selValueREALMax;
//		}
//		p->selValueREALOld = p->selValueREAL;
//		hmiParamListTableDisplayToValue(p->selValueREAL, p->listValuePtr[p->index], p->listValueText[p->index],
//			p->listDecPlaces[p->index], p->listLimits[p->index].k_factor, p->listLimits[p->index].n_factor, p->listLimits[p->index].valueType);
//	}
//
//	//keep checking if the source of the currently selected value changes on a PLC(i.e. PLC location gets updated, etc)
//	{
//		float tempVal = hmiParamListTableGetPLCValue(p->listValuePtr[p->index], p->listLimits[p->index].k_factor, p->listLimits[p->index].n_factor, p->listLimits[p->index].valueType);
//		if(p->selValueREAL != tempVal){
//			//PLC value changed > update displayed value
//			p->selValueREAL = tempVal;
//			p->selValueREALOld = p->selValueREAL;
//			hmiParamListTableDisplayToValue(p->selValueREAL, p->listValuePtr[p->index], p->listValueText[p->index],
//				p->listDecPlaces[p->index], p->listLimits[p->index].k_factor, p->listLimits[p->index].n_factor, p->listLimits[p->index].valueType);
//
//		}
//	}
//
//	//set default value request?
//	if(p->setDefaultRequest){
//		p->setDefaultRequest = 0;
//		p->selValueREAL = p->selValueREALDefault;
//	}
//
//}

//eof
```


- Program Logical/paiComponents/paiPing/paiPingService (ANSIC) (no source held here)

- Program Logical/paiComponents/paiUDP/udpApp (ANSIC) (no source held here)

### Package Logical/paiComponents/paiTemplate - pai Template Application with Drop down menues and tabs page navigation

### Package Logical/paiComponents/paiTemplate/paiHMI - Package

### paiHMI.typ - pai HMI types
```iecst
(********************************************************************
 * COPYRIGHT -- pai
 ********************************************************************
 * Package: HMI
 * File: HMI.typ
 * Author: goran
 * Created: August 28, 2013
 ********************************************************************
 * Data types of package HMI
 ********************************************************************)

TYPE
	hmiControlLogicEnums_typ :
		(
		hmiREMMEM_MAGIC := 16#55555555, (*Magic number*)
		hmiSecurityHMIUsersMAXIDX := 11, (*Max number of HMI users - 1*)
		hmiLoggerPVCmpBufSize := 2047, (*Size of the PV compare buffer*)
		HMI_PWD_LEVELS := 5, (*Number of password levels (0-operator;1-supervisor;2-admin;3-maintenance;4-factory)*)
		HMI_PWD_MAXLEN := 15 (*Max pwd len*)
		);
END_TYPE

(*########################################################################*)
(*Application object - Security Manager*)
(*########################################################################*)

TYPE
	hmiSecurityUser_typ : 	STRUCT
		loginLevel : UDINT; (*0-operator (no HMI access);1-supervisor;2-admin;3-maintenance;4-GAINCO*)
		userPIN : STRING[7];
		userName : STRING[63];
	END_STRUCT;
	hmiSecurityManager_typ : 	STRUCT
		webSecurityActive : UDINT;
		dbUpdateEvent : UDINT;
		visibleIfUserSecurityActive : UDINT;
		visibleIfUserSecurityNOTActive : UDINT;
		userIsLoggedIn : UDINT;
		loggedInUserIdx : UDINT;
		hmiUserIndex : UDINT;
		hmiUserIndexMax : UDINT;
		hmiPINSelected : UDINT;
		hmiPINCompletion : UDINT;
		hmiLoggedUserName : STRING[63];
		hmiListOfUserPINs : ARRAY[0..hmiSecurityHMIUsersMAXIDX]OF STRING[7];
		hmiListOfUserNames : ARRAY[0..hmiSecurityHMIUsersMAXIDX]OF STRING[63];
		listOfUsers : ARRAY[0..hmiSecurityHMIUsersMAXIDX]OF hmiSecurityUser_typ;
	END_STRUCT;
END_TYPE

(*########################################################################*)
(*Application object - Event Logger Manager*)
(*########################################################################*)

TYPE
	hmiEventLoggerManager_typ : 	STRUCT
		pvCompareEvent : UDINT; (*Set to 1 when MachineCfg strucutres changes. Allows logger manager to capture changed values and send them to DB.*)
		pvCompareResult : INT;
		pvCompareBuf : STRING[hmiLoggerPVCmpBufSize];
	END_STRUCT;
END_TYPE
```


- Data object Logical/acp10etxen (Ett) (no source held here)

### Package Logical/HMI - HMI screens 

### HMIremmem.typ - Global data types
```iecst
(********************************************************************
 * COPYRIGHT -- piedmont
 ********************************************************************
 * Package: HMI
 * File: HMIperm.typ
 * Author: goran
 * Created: August 28, 2013
 ********************************************************************
 * Data types of package HMI
 ********************************************************************)
(*########################################################################*)
(*HMI object - Remanent PV-s*)
(*########################################################################*)

TYPE
	hmiRemanent_typ : 	STRUCT
		magicNumber : UDINT; (*magic number to detect failure of the rem mem (i.e. drained battery)*)
	END_STRUCT;
	cfgRemanentData_typ : 	STRUCT  (*Configuration and recipe related data stored in remanent (battery backed) memory*)
		magicPrefix : UDINT; (*Set to 0x55555555 (MAGIC_NUMBER) to detect when/if battery backed memory changes*)
		magicPosfix : UDINT; (*Set to 0x55555555 (MAGIC_NUMBER) to detect when/if battery backed memory changes*)
	END_STRUCT;
END_TYPE
```

### Program Logical/HMI/hmilogic (ANSIC) - Service that manages navigating through the VC4 HMI

#### hmilogic.c
```c
/********************************************************************
 * COPYRIGHT -- piedmont
 ********************************************************************
 * Program: hmilogic
 * File: hmilogic.c
 * Author: goran
 * Created: August 28, 2013
 ********************************************************************
 * Implementation of program hmilogic
 ********************************************************************/

#include <bur/plctypes.h>

#ifdef _DEFAULT_INCLUDES
#include <AsDefault.h>
#endif

#include "hmiParamList.h"
#include "hmiDialog.h"
#include "hmiAlert.h"
#include "loginLogic_Header.h"

/*
###############################################################################
Utilities
###############################################################################
*/

/**
Bit manipulaiton utility functions.
 */
#include <../../bglib/bgBitUtilities.c>

#ifndef _BG_SPRINTF_H
#include <../../bglib/bgsprintf.h>
#include <../../bglib/bgsprintf.c>
#endif

#ifndef _BG_STRING_H
#include <../../bglib/bgstring.h>
#include <../../bglib/bgstring.c>
#endif

/*
###############################################################################
Menu keys logic
###############################################################################
*///logic control of the global MENU KEYS on the Left Side (i.e. STOPPED, FILLING, PRODUCTION, ...)
static void menuInitKeysLFRT()
{
	//make both menus not visible at the start
	gHmi.status.menuVisibleLT = 1;
	gHmi.status.menuVisibleRT = 1;
}

//logic control of the global MENU KEYS on the Left Side (i.e. STOPPED, FILLING, PRODUCTION, ...)
static void menuCyclicKeysRT()
{
	int ii;
	static UDINT menuVisibleLTOld;
	static UDINT menuVisibleRTOld;

	//make visible one of the 4 buttons stacked on each other
	//this is due to buttons are of different color and use border property to set the colors
	for(ii=0; ii<HMI_ENUM_MENU_ITEMS_RT;ii++){
		gHmi.status.menuVisibleRTItems[ii] = 1;
		if(ii == gHmi.status.menuIndexRT){
			gHmi.status.menuVisibleRTItems[ii] = 0;
		}
	}

	bgTimerCyclic(&gHmi.status.menuLFHideTimer);
	bgTimerCyclic(&gHmi.status.menuRTHideTimer);

	//when menu becomes visible > start the timer
	if(!gHmi.status.menuVisibleLT && menuVisibleLTOld){
		/*bgTimerStart(&gHmi.status.menuLFHideTimer, gConfig.active.hmi.dropdwMenuLFTimeout * 1000);*/ //dropdown timer LF
		bgTimerStart(&gHmi.status.menuLFHideTimer, DEFINE_MENU_L_HIDE_TIMEOUT_MS);
	}
	menuVisibleLTOld = gHmi.status.menuVisibleLT;
	//if menu still visible after timer expires > hide menu
	if( !gHmi.status.menuVisibleLT && bgTimerIsTimeOut(&gHmi.status.menuLFHideTimer) ){
		gHmi.status.menuVisibleLT = 1;
	}

	//when menu becomes visible > start the timer
	if(!gHmi.status.menuVisibleRT && menuVisibleRTOld){
		bgTimerStart(&gHmi.status.menuRTHideTimer, DEFINE_MENU_R_HIDE_TIMEOUT_MS); //dropdown timer LF
	}
	menuVisibleRTOld = gHmi.status.menuVisibleRT;
	//if menu still visible after timer expires > hide menu
	if( !gHmi.status.menuVisibleRT && bgTimerIsTimeOut(&gHmi.status.menuRTHideTimer) ){
		gHmi.status.menuVisibleRT = 1;
	}
}

/*
###############################################################################
Tab keys logic
###############################################################################
*///logic control of the tab key operation (i.e. radio button fuction)
static void menuInitTabKeys()
{
	//activate first tab (applies to any screen)
	gHmi.status.tabKeysRadioDataPoint = 1;
}

//logic control of the tab key operation (i.e. radio button fuction)
static void menuCyclicTabKeys()
{
	int ii;
	for(ii=0;ii<HMI_ENUM_TAB_KEYS_MAX;ii++){
		if(ii == gHmi.status.tabKeysRadioDataPoint){
			gHmi.status.tabKeysRadioArray[ii] = 1;//select array elements that matches selected radio button
		}else{
			gHmi.status.tabKeysRadioArray[ii] = 0;//unselect all other array elements
		}
	}
}

/*
###############################################################################
HMI screen handling logic
###############################################################################
*/
static void S_Global()
{
	menuCyclicKeysRT();
	menuCyclicTabKeys();
	loginLevelLogicCyclic();
}

//============================================================================
void screenHandlers(UINT page)
{
	hmiControlLogic_typ* pHmi = &gHmi;

	bgTimerCyclic(&gHmi.prv.tmr4);

	//Page specific init logic
	if(pHmi->prv.pageInit){
		//screen init event
		//define screen name
		switch(page){
			case HMI_HOME_10_DASHBOARD:
//				loginLevelParameterEditControl((UINT) gRecCfg.active.Cfg.HMI.Access_Level_HomeForce);
				break;
			case HMI_RECIPE_20_SELECT:
				loginLevelParameterEditControl(RECIPE_ACCESS_LEVEL);
				break;
			case HMI_CONFIG_30_SELECT:
				loginLevelParameterEditControl(CONFIG_ACCESS_LEVEL);
				break;
			case HMI_LOGIN_40_MAIN:
				bgStrCpyN(gHmi.status.passwordStrings[0], "0000", HMI_PWD_MAXLEN);
				bgStrCpyN(gHmi.status.passwordStrings[1], gRecCfg.active.Cfg.HMI.passwordSetup, HMI_PWD_MAXLEN);
				bgStrCpyN(gHmi.status.passwordStrings[2], gRecCfg.active.Cfg.HMI.passwordEngineer, HMI_PWD_MAXLEN);
				bgStrCpyN(gHmi.status.passwordStrings[3], gRecCfg.active.Cfg.HMI.passwordFactory, HMI_PWD_MAXLEN);
				break;
			case HMI_LOGIN_41_OPERATOR:
				break;
			case HMI_LOGIN_42_SETUP:
				break;
			case HMI_LOGIN_43_ENGINEER:

				break;
			case HMI_LOGIN_45_FACTORY:
				break;
			case HMI_MOTION_61_IO_MOTORS:
				loginLevelParameterEditControl(FORCEIO_ACCESS_LEVEL);
				break;
			case HMI_AUX_90_FILE:
//				loginLevelParameterEditControl(FORCEIO_ACCESS_LEVEL);
				break;
			default:
				strcpy(pHmi->prv.currentPageText, "screen() ????");
				break;
		}
	}

	if(pHmi->prv.pageExit){
		switch(page){
			default:
				break;
		}
	}

	//Page specific cyclic logic
	switch(page){
		case HMI_00_STARTUP:
			if( bgTimerIsTimeOut(&gHmi.prv.tmr4) ){
				gHmi.prv.changePage = HMI_HOME_10_DASHBOARD;
			}
			break;

		case HMI_RECIPE_21_PVLIST:
			break;

		case HMI_CONFIG_31_PVLIST:
			break;

		default:
			break;
	}

	//param table cyclic routine
	hmiParamListTableCyclic(&gHmiParamTable);
}

static void screenPageChangeLogic(hmiControlLogic_typ* pHmi)
{
	if(!pHmi)
		return;

	//operate screen logic timer
	bgTimerCyclic(&pHmi->prv.tmr1);

	//change screen is in progress; wait
	if(pHmi->prv.changePage != 0xFF)
		return;

	//generate page init/exit events
	pHmi->prv.pageInit = 0;
	pHmi->prv.pageExit = 0;
	if(pHmi->prv.currentPage != pHmi->prv.prevPage){
		pHmi->prv.pageExit = 1;
		screenHandlers(pHmi->prv.prevPage);
		pHmi->prv.pageExit = 0;

		pHmi->prv.pageInit = 1;
		pHmi->prv.prevPage = pHmi->prv.currentPage;

		//reset screen state
		pHmi->prv.state = 0;
		pHmi->prv.stateInit = 1;
	}else
		if(pHmi->prv.state != pHmi->prv.statePrev){

		//generate state init event
		pHmi->prv.statePrev = pHmi->prv.state;
		pHmi->prv.stateInit = 1;
	}
}
//============================================================================
static void screenLogicCyclic()
{
	hmiControlLogic_typ* pHmi = &gHmi;

	//Logic to detect page change events and generate approprite signals / flags (i/e/ pageInit etc)
	screenPageChangeLogic(pHmi);

	//Page(screen) specific logic. Logic that runs/applies only to a specific page/screen
	screenHandlers(pHmi->prv.currentPage);

	// TODO: S_Global() shall be possible to place above screenHandlers(). For now,
	//and due to clearing of one shot move related flags that's not working!!!!
	//Global screen logic that runs cyclicly
	S_Global();
}
//============================================================================

void _INIT hmilogicInit(void)
{

	gHmi.status.menuIndexLT = 0;

	menuInitKeysLFRT();
	menuInitTabKeys();
	hmiAlertHide(&gHmi.alertMsg);
	hmiDialogHide(&gHmi.dialogMsg);

	bgTimerStart(&gHmi.prv.tmr4, DEFINE_HMI_SPLASHSCREEN_TO_MS);
}
//============================================================================
void _CYCLIC hmilogicCyclic(void)
{

	screenLogicCyclic();

}
//============================================================================
```

- Visualisation Logical/HMI/VisuW1 (not shown)

### HMI_Page_Enum.typ - not listed in the package file held
```iecst
TYPE
	paiHMI_Page_Enum :
		(
		HMI_PAGE_00_CONNECTION_ERROR := 0,
		HMI_PAGE_01_MACHINE_SPLASH_PAGE := 1,
		HMI_PAGE_10_DASH_MAIN := 10,
		HMI_PAGE_20_PAR_CONFIG := 20,
		HMI_PAGE_21_PAR_RECIPE,
		HMI_PAGE_22_PAR_SAVE_LOAD,
		HMI_PAGE_23_PAR_IMPORT_EXPORT,
		HMI_PAGE_30_DIAG_ALERTS := 30,
		HMI_PAGE_31_DIAG_ALARMS,
		HMI_PAGE_32_DIAG_ALARM_HIST,
		HMI_PAGE_33_DIAG_APP_LOG,
		HMI_PAGE_40_HARDWARE_SDM := 40,
		HMI_PAGE_41_HARDWARE_SAFELOGIX,
		HMI_PAGE_42_HARDWARE_PANEL,
		HMI_PAGE_43_HARDWARE_NETWORK,
		HMI_PAGE_50_DATA_STATS := 50,
		HMI_PAGE_51_DATA_PV_TABLE,
		HMI_PAGE_52_DATA_PV_STATS,
		HMI_PAGE_53_DATA_OMAC_PACKML,
		HMI_PAGE_54_DATA_AUDIT,
		HMI_PAGE_55_DATA_OEE,
		HMI_PAGE_56_DATA_ENERGY,
		HMI_PAGE_57_DATA_ASSET_INTENSITY,
		HMI_PAGE_58_DATA_IMPORT_EXPORT,
		HMI_PAGE_60_ACCESS_LOGIN := 60,
		HMI_PAGE_61_ACCESS_USERS,
		HMI_PAGE_62_ACCESS_GROUPS,
		HMI_PAGE_63_ACCESS_IO,
		HMI_PAGE_70_MOTION_AXIS_SETUP := 70,
		HMI_PAGE_71_AXIS_MOVEMENT,
		HMI_PAGE_72_AXIS_TUNING,
		HMI_PAGE_73_AXIS_SERVICE,
		HMI_PAGE_80_MECHATRONICS_CNC := 80,
		HMI_PAGE_81_MECHATRONICS_DELTA,
		HMI_PAGE_82_MECHATRONICS_SPINDLE,
		HMI_PAGE_83_MECHATRONICS_TEACH,
		HMI_PAGE_84_MECHATRONICS_CAM,
		HMI_PAGE_90_USB_STATUS := 90,
		HMI_PAGE_91_USB_FILEIO
		);
END_TYPE
```

### RecCfg_Alarms.typ
```iecst
TYPE
	HERNON_Alarm_RecCfg_typ : 	STRUCT
		Belt_Length_Configuration_Error : BOOL; (*0*)
		Line_Scaling_Error : BOOL; (*1*)
		ACP_VCtrl_Scale_Error : BOOL; (*2*)
		App_SSI_Encoder_Config_Error : BOOL; (*3*)
		Invalid_Par_StartRequest : BOOL; (*4*)
		Invalid_Config_DispenseStart : BOOL; (*5*)
		Invalid_Config_InspectStart : BOOL; (*6*)
		Mechanics_Restart_Required : BOOL; (*7*)
		Default_Cfg_Set : BOOL; (*8*)
		Default_Rec_Set : BOOL; (*9*)
	END_STRUCT;
END_TYPE
```

### Program Logical/pkgRecCfg/Recipe_Handling (IEC)

#### Variables.var
```iecst
VAR
	pCmd : REFERENCE TO Recipe_HMI_Command_typ;
	loc_Timer_Find_Active : TON;
	ii_char : UDINT;
	locRefreshBeforeCall : BOOL;
	locDTGetTime : DTGetTime;
	locTimeString : STRING[255];
	locCurrentlySelectedCfgIsActive : USINT;
	locCurrentlySelectedRecIsActive : USINT;
	locFindActiveRecipe : USINT;
	ii_recipes : UINT;
	loc : Recipe_loc_typ := (0);
	pRecCfgUIConnect : REFERENCE TO MpRecipeUIConnectType;
END_VAR
(*Insert your comment here.*)
(*Insert your comment here.*)
(*Insert your comment here.*)
VAR
	Recipe_CSV_Control : MpRecipeCsv := (0);
	Recipe_CSV_Header : MpRecipeCsvHeaderType := (0);
	Recipe_CSV_RegPar : MpRecipeRegPar := (0);
	Recipe_CSV_UI : MpRecipeUI := (0);
	gRecipe_CSV_UIConnect : MpRecipeUIConnectType := (0);
END_VAR
(*Insert your comment here.*)
(*Insert your comment here.*)
VAR
	Config_CSV_Control : MpRecipeCsv := (0);
	Config_CSV_Header : MpRecipeCsvHeaderType := (0);
	Config_CSV_RegPar : MpRecipeRegPar := (0);
	Config_CSV_UI : MpRecipeUI := (0);
	gConfig_CSV_UIConnect : MpRecipeUIConnectType := (0);
END_VAR
(*Insert your comment here.*)
VAR
	Init_Logbook : FBK_Init_Logbook;
END_VAR
(*Insert your comment here.*)
```

#### Action_Set_Active_Rec.st
```iecst
ACTION Action_Set_Active_Rec:
//		FOR ii_recipes := 0 TO 19 BY 1 DO
//			IF (brsstrcmp(ADR(gRecipe_CSV_UIConnect.Recipe.List.Names[ii_recipes]), ADR(gRecipeName)) = 0) THEN
//				gRecipe_CSV_UIConnect.Recipe.List.SelectedIndex := ii_recipes;
//			END_IF;
//		END_FOR;

//	RETURN;

	gRecipe_CSV_UIConnect.Recipe.List.SelectedIndex := 0;

	FOR ii_recipes := 0 TO MAX_IDX_TOTAL_RECIPES BY 1 DO
		IF (brsstrcmp(ADR(gRecipe_CSV_UIConnect.Recipe.List.Names[gRecipe_CSV_UIConnect.Recipe.List.SelectedIndex]), ADR(gRecipeName)) = 0) THEN
			EXIT;
		ELSE
			gRecipe_CSV_UIConnect.Recipe.List.StepDown := 1;
			Recipe_CSV_UI();
		END_IF;
	END_FOR;

END_ACTION
```
